Omron CX-Programmer project NewProject (CX-Programmer 9.88)

# PLC AddOn_Final_Caulking: CJ2M CPU33
I/O table (CPU CJ2M-CPU33): rack 0 slot 11 CJ2M-EIP21

## Global symbols (name address type ; comment)
W463.00 BOOL  ; PB. dispenser ON
W56.00 BOOL  ; IND. dispenser On
3205.07 BOOL  ; CR Dispenser Oil ON
AL1 H400.00 BOOL  ; AL1_EMERGENCY STOP
AL10 H400.09 BOOL  ; AL10_AIR SOURCE PS. FAULT
AL100 H406.03 BOOL  ; AL100_AS.NG PULL FAULT
AL101 H406.04 BOOL  ; AL101_NG BOX FULL
AL102 H406.05 BOOL  ; AL102_WORK FINISH FULL
AL103 H406.06 BOOL  ; AL103_SAFET DOOR IS OPEN
AL104 H406.07 BOOL  ; AL104_Positioning TImeout
AL105 H406.08 BOOL  ; AL105_
AL106 H406.09 BOOL  ; AL106_
AL107 H406.10 BOOL  ; AL107_Oil Apply UD Fault
AL108 H406.11 BOOL  ; AL108_Oil Apply AR Fault
AL109 H406.12 BOOL  ; AL109_
AL11 H400.10 BOOL  ; AL11_DUMMY DOOR OPEN
AL110 H406.13 BOOL  ; AL110_
AL111 H406.14 BOOL  ; AL111_
AL112 H406.15 BOOL  ; AL112_
AL113 H407.00 BOOL  ; AL113_
AL114 H407.01 BOOL  ; AL114_
AL115 H407.02 BOOL  ; AL115_
AL116 H407.03 BOOL  ; AL116_
AL117 H407.04 BOOL  ; AL117_
AL118 H407.05 BOOL  ; AL118_
AL119 H407.06 BOOL  ; AL119_
AL12 H400.11 BOOL  ; AL12_SHUTTER DOOR INTERRUPTED
AL120 H407.07 BOOL  ; AL120_
AL121 H407.08 BOOL  ; AL121_
AL122 H407.09 BOOL  ; AL122_
AL123 H407.10 BOOL  ; AL123_
AL124 H407.11 BOOL  ; AL124
AL125 H407.12 BOOL  ; AL125_
AL126 H407.13 BOOL  ; AL126_
AL127 H407.14 BOOL  ; AL127_
AL128 H407.15 BOOL  ; AL128:
AL129 H408.00 BOOL  ; AL129:
AL13 H400.12 BOOL  ; AL13_FNCK EMERGENCY STOP
AL130 H408.01 BOOL  ; AL130:
AL131 H408.02 BOOL  ; AL131:
AL132 H408.03 BOOL  ; AL132:
AL133 H408.04 BOOL  ; AL133:
AL134 H408.05 BOOL  ; AL134:
AL135 H408.06 BOOL  ; AL135:
AL136 H408.07 BOOL  ; AL136:
AL137 H408.08 BOOL  ; AL137:
AL138 H408.09 BOOL  ; AL138:
AL139 H408.10 BOOL  ; AL139:
AL14 H400.13 BOOL  ; AL14_FNCK FUSE ABNORMAL
AL140 H408.11 BOOL  ; AL140:
AL141 H408.12 BOOL  ; AL141:
AL142 H408.13 BOOL  ; AL142:
AL143 H408.14 BOOL  ; AL143:
AL144 H408.15 BOOL  ; AL144:
AL145 H409.00 BOOL  ; AL145:
AL146 H409.01 BOOL  ; AL146:
AL147 H409.02 BOOL  ; AL147:
AL148 H409.03 BOOL  ; AL148:
AL149 H409.04 BOOL  ; AL149:
AL15 H400.14 BOOL  ; AL15_1EC1 ABNORMAL
AL150 H409.05 BOOL  ; AL150:
AL151 H409.06 BOOL  ; AL151:
AL152 H409.07 BOOL  ; AL152:
AL153 H409.08 BOOL  ; AL153:
AL154 H409.09 BOOL  ; AL154:
AL155 H409.10 BOOL  ; AL155:
AL156 H409.11 BOOL  ; AL156:
AL157 H409.12 BOOL  ; AL157:
AL158 H409.13 BOOL  ; AL158:
AL159 H409.14 BOOL  ; AL159:
AL16 H400.15 BOOL  ; AL16_1EC2 ABNORMAL
AL160 H409.15 BOOL  ; AL160:
AL161 H410.00 BOOL  ; AL161_PRODUCTION QUANTITY WARNING
AL162 H410.01 BOOL  ; AL162_DEFECT QUANTITY WARNING
AL163 H410.02 BOOL  ; AL163_TOTAL QUANTITY WARNING
AL164 H410.03 BOOL  ; AL164_
AL165 H410.04 BOOL  ; AL165_
AL166 H410.05 BOOL  ; AL166_
AL167 H410.06 BOOL  ; AL167_
AL168 H410.07 BOOL  ; AL168_
AL169 H410.08 BOOL  ; AL169:
AL17 H401.00 BOOL  ; AL17_1EC3 ABNORMAL
AL170 H410.09 BOOL  ; AL170_WIP DISCHARGE DONE
AL171 H410.10 BOOL  ; AL171_
AL172 H410.11 BOOL  ; AL172_
AL173 H410.12 BOOL  ; AL173_
AL174 H410.13 BOOL  ; AL174_
AL175 H410.14 BOOL  ; AL175_
AL176 H410.15 BOOL  ; AL176_
AL177 H411.00 BOOL  ; AL177_
AL178 H411.01 BOOL  ; AL178_
AL179 H411.02 BOOL  ; AL179_
AL18 H401.01 BOOL  ; AL18_1EC4 ABNORMAL
AL180 H411.03 BOOL  ; AL180_
AL181 H411.04 BOOL  ; AL181_
AL182 H411.05 BOOL  ; AL182_
AL183 H411.06 BOOL  ; AL183_
AL184 H411.07 BOOL  ; AL184_
AL185 H411.08 BOOL  ; AL185_
AL186 H411.09 BOOL  ; AL186_
AL187 H411.10 BOOL  ; AL187_
AL188 H411.11 BOOL  ; AL188_
AL189 H411.12 BOOL  ; AL189_
AL19 H401.02 BOOL  ; AL19_1MTD1 ABNORMAL
AL190 H411.13 BOOL  ; AL190_
AL191 H411.14 BOOL  ; AL191_
AL192 H411.15 BOOL  ; AL192_
AL193 H412.00 BOOL  ; AL193_
AL194 H412.01 BOOL  ; AL194_
AL195 H412.02 BOOL  ; AL195_
AL196 H412.03 BOOL  ; AL196:
AL197 H412.04 BOOL  ; AL197:
AL198 H412.05 BOOL  ; AL198:
AL199 H412.06 BOOL  ; AL199:
AL2 H400.01 BOOL  ; AL2_FUSE ABNORMAL
AL20 H401.03 BOOL  ; AL20:
AL200 H412.07 BOOL  ; AL200_PLC LOW BATTERY
AL201 H412.08 BOOL  ; AL201:
AL202 H412.09 BOOL  ; AL202:
AL203 H412.10 BOOL  ; AL203:
AL204 H412.11 BOOL  ; AL204:
AL205 H412.12 BOOL  ; AL205:
AL21 H401.04 BOOL  ; AL21:
AL22 H401.05 BOOL  ; AL22:
AL23 H401.06 BOOL  ; AL23:
AL24 H401.07 BOOL  ; AL24:
AL25 H401.08 BOOL  ; AL25:
AL26 H401.09 BOOL  ; AL26:
AL27 H401.10 BOOL  ; AL27:
AL28 H401.11 BOOL  ; AL28:
AL29 H401.12 BOOL  ; AL29:
AL3 H400.02 BOOL  ; AL3_SAFETY COVER OPEN
AL30 H401.13 BOOL  ; AL30:
AL31 H401.14 BOOL  ; AL31:
AL32 H401.15 BOOL  ; AL32:
AL33 H402.00 BOOL  ; AL33_CYCLE TIME OVER
AL34 H402.01 BOOL  ; AL34_FNCK MASTER OR AUTO STOP
AL35 H402.02 BOOL  ; AL35_FNCK FAULT OCCUR
AL36 H402.03 BOOL  ; AL36_MB LOADER 1 WORK LOST
AL37 H402.04 BOOL  ; AL37_MB LOADER 2 WORK LOST
AL38 H402.05 BOOL  ; AL38_POSITIONNING UNIT WORK LOST
AL39 H402.06 BOOL  ; AL39_TRANSFER SLIDE MB LOST
AL4 H400.03 BOOL  ; AL4_AIR SOURCE LOW
AL40 H402.07 BOOL  ; AL40_DIAPHAM LOADER 1 LOST WORK
AL41 H402.08 BOOL  ; AL41_DIAPHAM LOADER 2 LOST WORK
AL42 H402.09 BOOL  ; AL42_DIAPHAM LOADER 3 LOST WORK
AL43 H402.10 BOOL  ; AL43_DIAPHAM VACCUM STATION WORK LOST
AL44 H402.11 BOOL  ; AL44_DIAPHAM BUFFER STATION WORK LOST
AL45 H402.12 BOOL  ; AL45_DIAPHAM FEED IN STATION ABNORMAL
AL46 H402.13 BOOL  ; AL46_TRANFER SLIDE DIAPHAM LOST
AL47 H402.14 BOOL  ; AL47_ROTARY GRIPPER 1 LOST WORK
AL48 H402.15 BOOL  ; AL48_ROTARY GRIPPER 2 LOST WORK
AL49 H403.00 BOOL  ; AL49_WORK DISCHARGE UNIT WORK LOST
AL5 H400.04 BOOL  ; AL5_DEVICE-NET FAULT
AL50 H403.01 BOOL  ; AL50:Work Floating
AL51 H403.02 BOOL  ; AL51:
AL52 H403.03 BOOL  ; AL52:
AL53 H403.04 BOOL  ; AL53:
AL54 H403.05 BOOL  ; AL54:
AL55 H403.06 BOOL  ; AL55:
AL56 H403.07 BOOL  ; AL56:
AL57 H403.08 BOOL  ; AL57:
AL58 H403.09 BOOL  ; AL58:
AL59 H403.10 BOOL  ; AL59:
AL6 H400.05 BOOL  ; AL6_PLC ABNORMAL
AL60 H403.11 BOOL  ; AL60:
AL61 H403.12 BOOL  ; AL61:
AL62 H403.13 BOOL  ; AL62:
AL63 H403.14 BOOL  ; AL63:
AL64 H403.15 BOOL  ; AL64:
AL65 H404.00 BOOL  ; AL65_PRODUCTION QUANTITY UP
AL66 H404.01 BOOL  ; AL66_DEFECT QUANTITY UP
AL67 H404.02 BOOL  ; AL67_TOTAL QUANTITY UP
AL68 H404.03 BOOL  ; AL68_
AL69 H404.04 BOOL  ; AL69_
AL7 H400.06 BOOL
AL70 H404.05 BOOL  ; AL70_
AL71 H404.06 BOOL  ; AL71_
AL72 H404.07 BOOL  ; AL72_
AL73 H404.08 BOOL
AL74 H404.09 BOOL
AL75 H404.10 BOOL
AL76 H404.11 BOOL
AL77 H404.12 BOOL
AL78 H404.13 BOOL
AL79 H404.14 BOOL
AL8 H400.07 BOOL
AL80 H404.15 BOOL
AL81 H405.00 BOOL  ; AL81_AS.SHUTTER 1 FAULT
AL82 H405.01 BOOL  ; AL82_AS.SHUTTER 2 FAULT
AL83 H405.02 BOOL  ; AL83_AS.DIAPH GRIPPER UNIT FAULT
AL84 H405.03 BOOL  ; AL84_AS.DIAPH GRIPPER 1 FAULT
AL85 H405.04 BOOL  ; AL85_AS.DIAPH GRIPPER 2 FAULT
AL86 H405.05 BOOL  ; AL86_AS.DIAPH GRIPPER 3 FAULT
AL87 H405.06 BOOL  ; AL87_AS.DIAPH GRIPPER FLIP FAULT
AL88 H405.07 BOOL  ; AL88_AS.ROTARY GRIPPER 1 FAULT
AL89 H405.08 BOOL  ; AL89_AS.ROTARY GRIPPER 2 FAULT
AL9 H400.08 BOOL
AL90 H405.09 BOOL  ; AL90_AS.ROTARY GRIPPER UNIT 1 FAULT
AL91 H405.10 BOOL  ; AL91_AS.ROTARY GRIPPER UNIT 2 FAULT
AL92 H405.11 BOOL  ; AL92_AS.MB LOAD IN FAULT
AL93 H405.12 BOOL  ; AL93_AS.MB LOAD OUT FAULT
AL94 H405.13 BOOL  ; AL94_AS.MB LOAD OUT UNIT FAULT
AL95 H405.14 BOOL  ; AL95_AS.MB SLIDE UNIT FAULT
AL96 H405.15 BOOL  ; AL96_AS.MB POSITION PIN UNIT FAULT
AL97 H406.00 BOOL  ; AL97_AS.WORK TRANSFER UNIT FAULT
AL98 H406.01 BOOL  ; AL98_AS.FINISH TRAY FAULT
AL99 H406.02 BOOL  ; AL99_AS.OK PUSH FAULT
ALMF001 W501.00 BOOL  ; ALMF001_SHUTTER 1 OPERATION FAULT
ALMF002 W501.01 BOOL  ; ALMF002_SHUTTER 2 OPERATION FAULT
ALMF003 W501.02 BOOL  ; ALMF003_DIAPH GRIPPER UNIT OPERATION FAULT
ALMF004 W501.03 BOOL  ; ALMF004_DIAPH GRIPPER 1 OPERATION FAULT
ALMF005 W501.04 BOOL  ; ALMF005_DIAPH GRIPPER 2 OPERATION FAULT
ALMF006 W501.05 BOOL  ; ALMF006_DIAPH GRIPPER 3 OPERATION FAULT
ALMF007 W501.06 BOOL  ; ALMF007_DIAPH GRIPPER FLIP OPERATION FAULT
ALMF008 W501.07 BOOL  ; ALMF008_ROTARY GRIPPER 1 OPERATION FAULT
ALMF009 W501.08 BOOL  ; ALMF009_ROTARY GRIPPER 2 OPERATION FAULT
ALMF010 W501.09 BOOL  ; ALMF010_ROTARY GRIPPER UNIT 1 OPERATION FAULT
ALMF011 W501.10 BOOL  ; ALMF011_ROTARY GRIPPER UNIT 2 OPERATION FAULT
ALMF012 W501.11 BOOL  ; ALMF012_MB LOAD IN OPERATION FAULT
ALMF013 W501.12 BOOL  ; ALMF013_MB LOAD OUT OPERATION FAULT
ALMF014 W501.13 BOOL  ; ALMF014_MB LOAD OUT UNIT OPERATION FAULT
ALMF015 W501.14 BOOL  ; ALMF015_MB SLIDE UNIT OPERATION FAULT
ALMF016 W501.15 BOOL  ; ALMF016_MB POSITION PIN UNIT OPERATION FAULT
ALMF017 W502.00 BOOL  ; ALMF017_WORK TRANSFER UNIT OPERATION FAULT
ALMF018 W502.01 BOOL  ; ALMF018_FINISH TRAY OPERATION FAULT
ALMF019 W502.02 BOOL  ; ALMF019_OK PUSH OPERATION FAULT
ALMF020 W502.03 BOOL  ; ALMF020_NG PULL OPERATION FAULT
0.00 BOOL  ; PB.EMG STOP
0.01 BOOL  ; AIR SOURCE CONF.
0.02 BOOL  ; SS.AUTO-IND.(AUTO=ON)
0.03 BOOL  ; PB.MASTER ON
0.04 BOOL  ; PB.AUTO RUN
0.05 BOOL  ; PB.CYCLE STOP
0.06 BOOL  ; PB.DUMMY DOOR OPEN REQUEST
0.07 BOOL  ; CR.TEACHING ON
0.08 BOOL  ; CR.MACHINR DOOR CONFIRM
0.09 BOOL  ; CR.DUMMY DOOR CONFIRM
0.10 BOOL  ; CR.SHUTTER DOOR OUT CONFIRM
0.11 BOOL  ; CR.SHUTTER DOOR IN CONFIRM
0.12 BOOL  ; CR.MASTER ON CONFIRM
0.13 BOOL  ; CR.FUSE NORMAL CONFIRM
0.14 BOOL  ; CR.DIAPHAM DOOR ENABLE CONF
0.15 BOOL  ; .
1516 CHANNEL  ; SLAVE STATUS 1
1517 CHANNEL  ; SLAVE STATUS 2
1518 CHANNEL  ; SLAVE STATUS 3
1519 CHANNEL  ; SLAVE STATUS 4
1520 CHANNEL  ; NORMAL SLAVE1
1522 CHANNEL  ; NORMAL SLAVE3
1541 CHANNEL  ; SLAVE STATUS 1
1542 CHANNEL  ; SLAVE STATUS 2
1543 CHANNEL  ; SLAVE STATUS 3
1544 CHANNEL  ; SLAVE STATUS 4
1545 CHANNEL  ; NORMAL SLAVE STATUS 1
1547 CHANNEL  ; NORMAL SLAVE STATUS 3
1.00 BOOL  ; CR.EMERGENCY STOP INTERLOCK
1.01 BOOL  ; PL.AUTO RUNNING
1.02 BOOL  ; PL.MASTER ON
1.03 BOOL  ; PL.OK TO FEED DIAPHAM
1.04 BOOL  ; PL.DUMMY DOOR ENABLE CONFIRM
1.05 BOOL  ; PL.DUMMY PROCESS
1.06 BOOL  ; BZ.BUZZER
1.07 BOOL  ; CR.ADD-ON ABNORMAL INTERLOCK
1.08 BOOL  ; CR.ADD-ON AUTO RUN INTERLOCK
1.09 BOOL  ; CR.DUMMY DOOR ENABLE TO OPEN
1.10 BOOL  ; CR Interupt Safety area
1.11 BOOL  ; CR.TEACHING ENABLE
1.12 BOOL  ; CR.ADD-ON AUTO START
1.13 BOOL  ; PL.SIGNAL TOWER R
1.14 BOOL  ; PL.SIGNAL TOWER Y
1.15 BOOL  ; PL.SIGNAL TOWER G
2.00 BOOL  ; ITLK.PB FINAL EMERGENCY NOT
2.01 BOOL  ; ITLK.FINAL CAULKING FUSE CONFIRM
2.02 BOOL  ; ITLK.FINAL CAULKING-MASTER ON,AUTO RUNNING
2.03 BOOL  ; ITLK.FINAL CAULKING-ALL HOME
2.04 BOOL  ; ITLK.FINAL CAULKING DIAPH BLOW OK
2.05 BOOL  ; ITLK.FINAL CAULKING ABNORMAL DETECTION
2.06 BOOL  ; .
2.07 BOOL  ; ITLK.FINAL CAULKING-AUTO M&B VACCUM OK
2.08 BOOL  ; ITLK.FINAL CAULKING-AUTO DIAPH VACCUM OK
2.09 BOOL  ; ITLK.FINAL CAULKING WORK OK
2.10 BOOL  ; ITLK.FINAL CAULKING WORK NG
2.11 BOOL  ; ITLK.FINAL CAULKING WORK OPERATE
2.12 BOOL  ; ITLK.PH FINAL CAULKING ST1 DETECT
2.13 BOOL  ; ITLK.PH FINAL CAULKING ST2 DETECT
2.14 BOOL  ; .
2.15 BOOL  ; .
3205.00 BOOL  ; 1MTD1.FWD
3205.01 BOOL  ; 1MTD1.REV
3205.02 BOOL  ; 1MTD1.MO
3205.03 BOOL  ; 1MGH1 START
3205.04 BOOL  ; 1MGH1 STOP
3205.05 BOOL  ; 1MGH2 START
3205.06 BOOL  ; 1MGH2 STOP
3205.08 BOOL  ; SOL. SHUTTER DOOR 1 DOWN
3205.09 BOOL  ; SOL. SHUTTER DOOR 2 UP
3205.10 BOOL  ; SOL. SHUTTER DOOR 2 DOWN
3205.15 BOOL  ; PL.LOAD WORK ENABLE
3207.00 BOOL  ; SOL_Oil Apply Ret
3207.01 BOOL  ; SOL_Oil Apply Adv
3207.02 BOOL  ; SOL_Oil Apply Down
3207.03 BOOL  ; SOL_Oil Apply Up
3211.00 BOOL  ; M&B LOAD UNIT SLIDE ADV
3211.01 BOOL  ; M&B LOAD UNIT SLIDE RET
3211.02 BOOL  ; M&B LOAD IN DOWN
3211.03 BOOL  ; M&B LOAD IN UP
3211.04 BOOL  ; M&B LOAD OUT UNIT DOWN
3211.05 BOOL  ; M&B LOAD OUT UNIT UP
3211.06 BOOL  ; M&B LOAD OUT DOWN
3211.07 BOOL  ; M&B LOAD OUT UP
3211.08 BOOL  ; PIN POSIRIONNING UP
3211.09 BOOL  ; PIN POSIRIONNING DOWN
3211.10 BOOL  ; NG PUSH DOWN
3211.11 BOOL  ; NG PUSH UP
3211.12 BOOL  ; OK PUSH UP
3211.13 BOOL  ; OK PUSH DOWN
3211.14 BOOL  ; LOAD BWD
3211.15 BOOL  ; LOAD FWD
3213.00 BOOL  ; WORK FINISH TRAY DOWN CONFIRM
3213.01 BOOL  ; WORK FINISH TRAY UP CONFIrM
3213.02 BOOL  ; TRANSFER SLIDE UNIT ADV
3213.03 BOOL  ; TRANSFER SLIDE UNIT RET
3213.04 BOOL  ; GIPPER TRANSFER UNIT 1 UNIT ADV
3213.05 BOOL  ; GIPPER TRANSFER UNIT 1 UNIT RET
3213.06 BOOL  ; GIPPER TRANSFER UNIT 2 UNIT ADV
3213.07 BOOL  ; GIPPER TRANSFER UNIT 2 UNIT RET
3213.08 BOOL  ; GIPPER TRANSFER 1 UNIT CHUCK
3213.09 BOOL  ; GIPPER TRANSFER 1 UNIT UNCHUCK
3213.10 BOOL  ; GIPPER TRANSFER 2 UNIT CHUCK
3213.11 BOOL  ; GIPPER TRANSFER 2 UNIT UNCHUCK
3213.12 BOOL  ; .
3213.13 BOOL  ; .
3213.14 BOOL  ; .
3213.15 BOOL  ; .
3215.00 BOOL  ; GRIPPER UNIT DOWN
3215.01 BOOL  ; GRIPPER UNIT UP
3215.02 BOOL  ; GRIPPER 1 DIAPH CHUCK
3215.03 BOOL  ; GRIPPER 1 DIAPH UNCHUCK
3215.04 BOOL  ; GRIPPER 2 DIAPH CHUCK
3215.05 BOOL  ; GRIPPER 2 DIAPH UNCHUCK
3215.06 BOOL  ; FLIP DIAPH 180
3215.07 BOOL  ; FLIP DIAPH 0
3215.08 BOOL  ; GRIPPER 3 DIAPH CHUCK
3215.09 BOOL  ; GRIPPER 3 DIAPH UNCHUCK
3215.10 BOOL  ; .
3215.11 BOOL  ; .
3215.12 BOOL  ; .
3215.13 BOOL  ; .
3215.14 BOOL  ; .
3215.15 BOOL  ; .
3301.00 BOOL  ; AS.SHUTTER 1 DOOR UP CONFIRM
3301.01 BOOL  ; AS.SHUTTER 1 DOOR DOWN CONFIRM
3301.02 BOOL  ; AS.SHUTTER 2 DOOR UP CONFIRM
3301.03 BOOL  ; AS.SHUTTER 2 DOOR DOWN CONFIRM
3301.04 BOOL  ; AS.GRIPPER UNIT DOWN CONFIRM
3301.05 BOOL  ; AS.GRIPPER UNIT UP CONFIRM
3301.06 BOOL  ; AS.GRIPPER 1 DIAPH CHUCK. CONFIRM
3301.07 BOOL  ; AS.GRIPPER 1 DIAPH UNCHUCK. CONFIRM
3301.08 BOOL  ; AS.GRIPPER 2 DIAPH CHUCK. CONFIRM
3301.09 BOOL  ; AS.GRIPPER 2 DIAPH UNCHUCK. CONFIRM
3301.10 BOOL  ; AS.GRIPPER 3 DIAPH CHUCK. CONFIRM
3301.11 BOOL  ; AS.GRIPPER 3 DIAPH UNCHUCK. CONFIRM
3301.12 BOOL  ; AS.FLIP DIAPH 180. CONFIRM
3301.13 BOOL  ; AS.FLIP DIAPH 0. CONFIRM
3301.14 BOOL  ; 1MTD1.ALARM
3301.15 BOOL  ; AUTO START(NAGARA)
3302.00 BOOL  ; AS.GIPPER TRANSFER 1 UNIT CHUCK CONFIRM
3302.01 BOOL  ; AS.GIPPER TRANSFER 1 UNIT  UNCHUCK CONFIRM
3302.02 BOOL  ; AS.GIPPER TRANSFER 2 UNIT CHUCK CONFIRM
3302.03 BOOL  ; AS.GIPPER TRANSFER 2 UNIT  UNCHUCK CONFIRM
3302.04 BOOL  ; AS.GIPPER TRANSFER UNIT 1 UNIT ADV. CONFIRM
3302.05 BOOL  ; AS.GIPPER TRANSFER UNIT 1 UNIT RET. CONFIRM
3302.06 BOOL  ; AS.GIPPER TRANSFER UNIT 2 UNIT ADV. CONFIRM
3302.07 BOOL  ; AS.GIPPER TRANSFER UNIT 2 UNIT RET. CONFIRM
3302.08 BOOL  ; PH MB VAcuum
3302.09 BOOL  ; PH. WORK FULL
3302.10 BOOL  ; PH.TRANSFER STATION DIAPH SIDE CONFIRM
3302.11 BOOL  ; PH.TRANSFER STATION DIAPH WORK CONFIRM
3302.12 BOOL  ; PH.TRANSFER STATION M&B WORK CONFIRM
3302.13 BOOL  ; PH. M&B LOADER WORK CONF 1
3302.14 BOOL  ; PH. M&B LOADER WORK CONF 2
3302.15 BOOL  ; PH. WORK IN ROTATE UNIT CONFIRM
3303.00 BOOL  ; AS.M&B LOAD IN DOWN.CONFIRM
3303.01 BOOL  ; AS.M&B LOAD IN UP.CONFIRM
3303.02 BOOL  ; AS.M&B LOAD OUT DOWN.CONFIRM
3303.03 BOOL  ; AS.M&B LOAD OUT UP.CONFIRM
3303.04 BOOL  ; AS.M&B LOAD OUT UNIT DOWN.CONFIRM
3303.05 BOOL  ; AS.M&B LOAD OUT UNIT UP.CONFIRM
3303.06 BOOL  ; AS.M&B LOAD UNIT SLIDE ADV.CONFIRM
3303.07 BOOL  ; AS.M&B LOAD UNIT SLIDE RET.CONFIRM
3303.08 BOOL  ; AS.PIN POSIRIONNING UP CONFIRM
3303.09 BOOL  ; AS.PIN POSIRIONNING DOWN CONFIRM
3303.10 BOOL  ; AS.TRANSFER SLIDE UNIT ADV. CONFIRM
3303.11 BOOL  ; AS.TRANSFER SLIDE UNIT RET. CONFIRM
3303.12 BOOL  ; PH work infinish tray
3303.13 BOOL  ; .
3303.14 BOOL  ; AS LOAD BWD
3303.15 BOOL  ; AS LOAD FWD
3304.00 BOOL  ; AS.WORK FINISH TRAY DOWN CONFIRM
3304.01 BOOL  ; AS.WORK FINISH TRAY UP CONFIRM
3304.02 BOOL  ; AS.OK PUSH UP. CONFIRM
3304.03 BOOL  ; AS.OK PUSH DOWN. CONFIRM
3304.04 BOOL  ; AS.NG PUSH DOWN. CONFIRM
3304.05 BOOL  ; AS.NG PUSH UP. CONFIRM
3304.06 BOOL  ; .
3304.07 BOOL  ; temporary nagara
3304.08 BOOL  ; PH. WORK ROTATE PRE-END CONFIRM
3304.09 BOOL  ; PH. TEMINAL IN POSITION CONFIRM
3304.10 BOOL  ; PH. WORK DIAPH LOAD IN CONFIRM
3304.11 BOOL  ; PH.STATION DIAPH VACCUM CONFIRM
3304.12 BOOL  ; PH.STATION BUFFER DIAPH CONFIRM
3304.13 BOOL  ; PH. WORK NG CONFIRM
3304.14 BOOL  ; PH. WORK OK CONFIRM
3304.15 BOOL  ; Safety AREA
3307.00 BOOL  ; RS_Oil Apply DOWN
3307.01 BOOL  ; RS_Oil Apply UP
3307.02 BOOL  ; RS_Oil Apply ADV
3307.03 BOOL  ; RS_Oil Apply RET
3334.01 BOOL  ; AS.WORK FINISH TRAY UP CONFIRM
3356.01 BOOL  ; diap auto
370.10 BOOL  ; PL HMI CAULKING ST1
370.11 BOOL  ; PL Rotary Gipper 2
370.12 BOOL  ; PL rotary gripper 1
370.13 BOOL  ; PL OKNG disch
3.00 BOOL  ; 1EC1.FORWARD START (DOWN)
3.01 BOOL  ; 1EC1.BACKWARD START (UP)
3.02 BOOL  ; 1EC1.ALARM RESET
3.03 BOOL  ; 1EC1.BREAK RELEASE (MTN)
3.04 BOOL  ; 1EC2.FWD START
3.05 BOOL  ; 1EC2.BWD START
3.06 BOOL  ; 1EC2.ALARM RESET
3.07 BOOL  ; 1EC2.BREAK RELEASE (MTN)
3.08 BOOL  ; 1EC3.FORWARD START
3.09 BOOL  ; 1EC3.BACKWARD START
3.10 BOOL  ; 1EC3.ALARM RESET
3.11 BOOL  ; 1EC3.BREAK RELEASE (MTN)
3.12 BOOL  ; 1EC4.FORWARD START
3.13 BOOL  ; 1EC4.BACKWARD START
3.14 BOOL  ; 1EC4.ALARM RESET
3.15 BOOL  ; 1EC4.BREAK RELEASE (MTN)
4450.00 BOOL  ; PB triall mode
4460.00 BOOL  ; PL trial mode
4.00 BOOL  ; 1EC1.FORWARD COMPLETE
4.01 BOOL  ; 1EC1.BACKWARD COMPLETE
4.02 BOOL  ; 1EC1.ALARM
4.03 BOOL  ; 1EC2.FORWARD COMPLETE
4.04 BOOL  ; 1EC2.BACKWARD COMPLETE
4.05 BOOL  ; 1EC2.ALARM
4.06 BOOL  ; 1EC3.FORWARD COMPLETE
4.07 BOOL  ; 1EC3.BACKWARD COMPLETE
4.08 BOOL  ; 1EC3.MIDDLE COMPLETE
4.09 BOOL  ; .
4.10 BOOL  ; .
4.11 BOOL  ; 1EC4.BACKWARD COMPLETE
4.12 BOOL  ; 1EC4.ALARM
4.15 BOOL  ; Safety area
56.06 BOOL  ; TIMER
5.00 BOOL  ; DIAPHAM DOOR ENABLE
5.01 BOOL  ; IAI EC POWER
5.05 BOOL  ; MG1 ON
5.06 BOOL  ; mg 1 off
5.07 BOOL  ; mg 2 on
5.08 BOOL  ; mg2 off
999.00 BOOL  ; ASAKE MODIFY (Oil Apply)
A202.00 BOOL  ; Communications Port Enabled Flag, Port No. 0
A202.01 BOOL  ; Communications Port Enabled Flag, Port No. 1
A202.02 BOOL  ; Communications Port Enabled Flag, Port No. 2
A202.03 BOOL  ; Communications Port Enabled Flag, Port No. 3
A202.04 BOOL  ; Communications Port Enabled Flag, Port No. 4
A202.05 BOOL  ; Communications Port Enabled Flag, Port No. 5
A202.06 BOOL  ; Communications Port Enabled Flag, Port No. 6
A202.07 BOOL  ; Communications Port Enabled Flag, Port No. 7
A401.10 BOOL  ; I/O_SETTING FAULT FLAG
A401.11 BOOL  ; I/O_MARK OVER FLAG
A401.13 BOOL  ; No.DOBLE USE FAULT FLAG
A401.14 BOOL  ; I/O BUS FAULT FLAG
A401.15 BOOL  ; MEMORY FAULT FLAG
A402.02 BOOL  ; High performance I/O unit setting and abnormality flags
A402.03 BOOL  ; CPU high performance unit setting and abnormality flags
A402.07 BOOL  ; High performance I unit of CPU abnormal flag
C0401 BOOL  ; CT01_LOW_UP
C0402 BOOL  ; CT01_HI_UP
C0403 BOOL  ; CT02_LOW_UP
C0404 BOOL  ; CT02_HI_UP
C0405 BOOL  ; CT03_LOW_UP
C0406 BOOL  ; CT03_HI_UP
C0407 BOOL  ; CT04_LOW_UP
C0408 BOOL  ; CT04_HI_UP
C0409 BOOL  ; CT05_LOW_UP
C0410 BOOL  ; CT05_HI_UP
C0411 BOOL  ; CT06_LOW_UP
C0412 BOOL  ; CT06_HI_UP
C0413 BOOL  ; CT07_LOW_UP
C0414 BOOL  ; CT07_HI_UP
C0415 BOOL  ; CT08_LOW_UP
C0416 BOOL  ; CT08_HI_UP
C0417 BOOL  ; CT09_LOW_UP
C0418 BOOL  ; CT09_HI_UP
C0419 BOOL  ; CT10_LOW_UP
C0420 BOOL  ; CT10_HI_UP
C0421 BOOL  ; CT11_LOW_UP
C0422 BOOL  ; CT11_HI_UP
C0423 BOOL  ; CT12_LOW_UP
C0424 BOOL  ; CT12_HI_UP
C0425 BOOL  ; CT13_LOW_UP
C0426 BOOL  ; CT13_HI_UP
C0427 BOOL  ; CT14_LOW_UP
C0428 BOOL  ; CT14_HI_UP
C0429 BOOL  ; CT15_LOW_UP
C0430 BOOL  ; CT15_HI_UP
C0451 BOOL  ; T1_LOW_UP
C0453 BOOL  ; T2_LOW_UP
C0455 BOOL  ; T3_LOW_UP
C0457 BOOL  ; T4_LOW_UP
C0459 BOOL  ; T5_LOW_UP
C0461 BOOL  ; T6_LOW_UP
C0468 BOOL  ; MONITORING CT_LOW
C0472 BOOL  ; AUTOMATIC TIME S
C0473 BOOL  ; AUTOMATIC TIME M
C0474 BOOL  ; AUTOMATIC TIME H
C0475 BOOL  ; WAITING-TIME S
C0476 BOOL  ; WAITING-TIME M
C0478 BOOL  ; STOP TIME S
C0479 BOOL  ; STOP TIME M
C0501 BOOL  ; OUTPUT 1 CUMULATE TIME m
C0502 BOOL  ; OUTPUT 2 CUMULATE TIME m
C0503 BOOL  ; OUTPUT 3 CUMULATE TIME m
C0504 BOOL  ; OUTPUT 4 CUMULATE TIME m
C0505 BOOL  ; OUTPUT 5 CUMULATE TIME m
C401 CHANNEL  ; CT01_LOW
C402 CHANNEL  ; CT01_HI
C403 CHANNEL  ; CT02_LOW
C404 CHANNEL  ; CT02_HI
C405 CHANNEL  ; CT03_LOW
C406 CHANNEL  ; CT03_HI
C407 CHANNEL  ; CT04_LOW
C408 CHANNEL  ; CT04_HI
C409 CHANNEL  ; CT05_LOW
C410 CHANNEL  ; CT05_HI
C411 CHANNEL  ; CT06_LOW
C412 CHANNEL  ; CT06_HI
C413 CHANNEL  ; CT07_LOW
C414 CHANNEL  ; CT07_HI
C415 CHANNEL  ; CT08_LOW
C416 CHANNEL  ; CT08_HI
C417 CHANNEL  ; CT09_LOW
C418 CHANNEL  ; CT09_HI
C419 CHANNEL  ; CT10_LOW
C420 CHANNEL  ; CT10_HI
C421 CHANNEL  ; CT11_LOW
C422 CHANNEL  ; CT11_HI
C423 CHANNEL  ; CT12_LOW
C424 CHANNEL  ; CT12_HI
C425 CHANNEL  ; CT13_LOW
C426 CHANNEL  ; CT13_HI
C427 CHANNEL  ; CT14_LOW
C428 CHANNEL  ; CT14_HI
C429 CHANNEL  ; CT15_LOW
C430 CHANNEL  ; CT15_HI
C451 CHANNEL  ; T1_LOW
C452 CHANNEL  ; T1_HI
C453 CHANNEL  ; T2_LOW
C454 CHANNEL  ; T2_HI
C455 CHANNEL  ; T3_LOW
C456 CHANNEL  ; T3_HI
C457 CHANNEL  ; T4_LOW
C458 CHANNEL  ; T4_HI
C459 CHANNEL  ; T5_LOW
C460 CHANNEL  ; T5_HI
C461 CHANNEL  ; T6_LOW
C462 CHANNEL  ; T6_HI
C501 CHANNEL  ; OUTPUT 1 CUMULATE TIME m
C502 CHANNEL  ; OUTPUT 2 CUMULATE TIME m
C503 CHANNEL  ; OUTPUT 3 CUMULATE TIME m
C504 CHANNEL  ; OUTPUT 4 CUMULATE TIME m
C505 CHANNEL  ; OUTPUT 5 CUMULATE TIME m
D1 CHANNEL  ; MB Loader Work Grip
D100 CHANNEL  ; SUM MB AUX1
D101 CHANNEL  ; SUM ALL MB
D110 CHANNEL  ; AUX1
D111 CHANNEL  ; AUX2
D112 CHANNEL  ; AUX3
D113 CHANNEL  ; WORK DIAPHAM +1
D114 CHANNEL  ; DIAPH SUMMARY
D12 CHANNEL  ; MB Rotate Work
D200 CHANNEL  ; WORK LAST ORER
D2000 CHANNEL  ; MB LOAD IN TIMER
D201 CHANNEL  ; WORK FEED OUT
D202 CHANNEL  ; LAST ORDER COUNT FOR P16
D22 CHANNEL  ; TRANSFER WORK
D23 CHANNEL  ; TRANSFER WORK
D3000 CHANNEL  ; DATA PASSWORD FROM SREEN
D3004 CHANNEL  ; DATA PASS WORD CHECK USE
D3020 CHANNEL  ; OFFSET ANGLE HMI
D3024 CHANNEL  ; OFFSET ANGLE USE
D3030 CHANNEL  ; DATA ANGLE NEW OFFSET
D32 CHANNEL  ; WORK FEED IN
D3500 CHANNEL  ; DATA MM/DD (HEX)
D3502 CHANNEL  ; DATA YYYY (HEX)
D3504 CHANNEL  ; DATA MM/DD (ASC)
D3512 CHANNEL  ; DATA YYYY ASCII
D3520 CHANNEL  ; DATA YYYY(ASCII)
D4000 CHANNEL  ; No.WORD SUM CHECK
D4001 CHANNEL  ; CONTROL DATA 2
D41 CHANNEL  ; DPH Loader GRIP
D4100 CHANNEL  ; TOURQE CHECK +NG
D4102 CHANNEL  ; TOURQE CHECK -NG
D4104 CHANNEL  ; ANGLE CHECK +NG
D4106 CHANNEL  ; ANGLE CHECK -NG
D42 CHANNEL  ; DPH Loader BUFF
D5000 CHANNEL  ; VT PAGE MONITOR
D5002 CHANNEL  ; VT PAGE CONTROL
D5003 CHANNEL  ; VT SCREEN ON-OFF
D5006 CHANNEL  ; OPERATION MONITORING OUTPUT
D5011 CHANNEL  ; OPERATION MONITORING TRANSMISSION
D5013 CHANNEL  ; OPERATION MONITORING TRANSMISSION
D5047 CHANNEL  ; COMPLETED CHECK
D5049 CHANNEL  ; WATCH_DOG_HEXFF
D5066 CHANNEL  ; CYCLE TIME
D5100 CHANNEL  ; CYCLE TIME SETTING (LOW RANK)
D5101 CHANNEL  ; ACTIVE-TIME H SETTING (LOW RANK)
D5102 CHANNEL  ; ACTIVE-TIME M SETTING (LOW RANK)
D5103 CHANNEL  ; PLAN TIME H SETTING (LOW RANK)
D5104 CHANNEL  ; PLAN TIME M SETTING (LOW RANK)
D5105 CHANNEL  ; QUANTITY (LOW RANK)
D5106 CHANNEL  ; QUANTITY (HIGHER RANK)
D5108 CHANNEL  ; AUTOMATIC TIME M
D5109 CHANNEL  ; AUTOMATIC TIME H
D5111 CHANNEL  ; WAITING-TIME M
D5113 CHANNEL  ; STOP TIME M
D5120 CHANNEL  ; FAULT CHECK
D5121 CHANNEL  ; MOTION FAULT CHECK
D5131 CHANNEL  ; CT01 COUNTER
D5133 CHANNEL  ; CT02 COUNTER
D5135 CHANNEL  ; CT03 COUNTER
D5137 CHANNEL  ; CT04 COUNTER
D5139 CHANNEL  ; CT05 COUNTER
D5141 CHANNEL  ; CT06 COUNTER
D5143 CHANNEL  ; CT07 COUNTER
D5145 CHANNEL  ; CT08 COUNTER
D5147 CHANNEL  ; CT09 COUNTER
D5149 CHANNEL  ; CT10 COUNTER
D5151 CHANNEL  ; CT11 COUNTER
D5153 CHANNEL  ; CT12 COUNTER
D5155 CHANNEL  ; CT13 COUNTER
D5157 CHANNEL  ; CT14 COUNTER
D5159 CHANNEL  ; CT15 COUNTER
D5231 CHANNEL  ; CT01 COUNTER
D5341 CHANNEL  ; OUTPUT 1 START DELAY TIME
D5342 CHANNEL  ; OUTPUT 2 START DELAY TIME
D5343 CHANNEL  ; OUTPUT 3 START DELAY TIME
D5344 CHANNEL  ; OUTPUT 4 START DELAY TIME
D5345 CHANNEL  ; OUTPUT 5 START DELAY TIME
D5351 CHANNEL  ; OUTPUT 1 BREAK DELAY TIME
D5352 CHANNEL  ; OUTPUT 2 BREAK DELAY TIME
D5353 CHANNEL  ; OUTPUT 3 BREAK DELAY TIME
D5354 CHANNEL  ; OUTPUT 4 BREAK DELAY TIME
D5355 CHANNEL  ; OUTPUT 5 BREAK DELAY TIME
D5461 CHANNEL  ; OUTPUT 1 STOP SELECTION
D5462 CHANNEL  ; OUTPUT 2 STOP SELECTION
D5463 CHANNEL  ; OUTPUT 3 STOP SELECTION
D5464 CHANNEL  ; OUTPUT 4 STOP SELECTION
D5465 CHANNEL  ; OUTPUT 5 STOP SELECTION
D5471 CHANNEL  ; OUTPUT 1 EXTERNAL PRESENCE SEL.
D5472 CHANNEL  ; OUTPUT 2 EXTERNAL PRESENCE SEL.
D5473 CHANNEL  ; OUTPUT 3 EXTERNAL PRESENCE SEL.
D5474 CHANNEL  ; OUTPUT 4 EXTERNAL PRESENCE SEL.
D5475 CHANNEL  ; OUTPUT 5 EXTERNAL PRESENCE SEL.
D5481 CHANNEL  ; OUTPUT 1 LOW ENERGY TIME
D5482 CHANNEL  ; OUTPUT 2 LOW ENERGY TIME
D5483 CHANNEL  ; OUTPUT 3 LOW ENERGY TIME
D5484 CHANNEL  ; OUTPUT 4 LOW ENERGY TIME
D5485 CHANNEL  ; OUTPUT 5 LOW ENERGY TIME
D5486 CHANNEL  ; OUTPUT 1 START DELAY TIME(BIN)
D5487 CHANNEL  ; OUTPUT 2 START DELAY TIME(BIN)
D5488 CHANNEL  ; OUTPUT 3 START DELAY TIME(BIN)
D5489 CHANNEL  ; OUTPUT 4 START DELAY TIME(BIN)
D5490 CHANNEL  ; OUTPUT 5 START DELAY TIME(BIN)
D5491 CHANNEL  ; OUTPUT 1 LOW ENERGY TIME(BIN)
D5492 CHANNEL  ; OUTPUT 2 LOW ENERGY TIME(BIN)
D5493 CHANNEL  ; OUTPUT 3 LOW ENERGY TIME(BIN)
D5494 CHANNEL  ; OUTPUT 4 LOW ENERGY TIME(BIN)
D5495 CHANNEL  ; OUTPUT 5 LOW ENERGY TIME(BIN)
D5496 CHANNEL  ; OUTPUT 1 BREAK DELAY TIME(BIN)
D5497 CHANNEL  ; OUTPUT 2 BREAK DELAY TIME(BIN)
D5498 CHANNEL  ; OUTPUT 3 BREAK DELAY TIME(BIN)
D5499 CHANNEL  ; OUTPUT 4 BREAK DELAY TIME(BIN)
D5500 CHANNEL  ; OUTPUT 5 BREAK DELAY TIME(BIN)
D5600 CHANNEL  ; WORK INFO
D6000 CHANNEL  ; FIRST ID DATA READ
D6003 CHANNEL  ; SUM CHECK
D6004 CHANNEL  ; SOURCE FIRST DATA
D6006 CHANNEL  ; SERAIL No. FROM ID
D6008 CHANNEL  ; PART No. FROM ID
D6009 CHANNEL  ; PROCESS COMPLETE 1 READ FORM ID
D6010 CHANNEL  ; PROCESS COMPLETE MC.No.2 READ FORM ID
D6011 CHANNEL  ; PROCESS OK 1 FROM ID
D6013 CHANNEL  ; WORK INFO
D6031 CHANNEL  ; FINAL ID DATA READ
D6205 CHANNEL  ; TORQUE DATA 1st STAGE (ARRANGED)
D6206 CHANNEL  ; ANGLE DATA 1st STAGE (ARRANGED)
D6207 CHANNEL  ; SNUG TORQUE 1st STAGE (ARRANGED)
D6208 CHANNEL  ; TORQUE DATA 2nd STAGE (ARRANGED)
D6209 CHANNEL  ; ANGLE DATA 2nd STAGE (ARRANGED)
D6210 CHANNEL  ; SNUG TORQUE 2nd STAGE (ARRANGED)
D6211 CHANNEL  ; T/R1 2nd STAGE (ARRANGED)
D6212 CHANNEL  ; T/R2 2nd STAGE (ARRANGED)
D6213 CHANNEL  ; BT/R 2nd STAGE (ARRANGED)
D6220 CHANNEL  ; STAGE DATA
D6500 CHANNEL  ; START INDEX MEMORY
D6502 CHANNEL  ; INDEX MEMORY PARAMETER
D6510 CHANNEL  ; MODEL USED
D6520 CHANNEL  ; PLUG RELIEF SIDE USED
D6521 CHANNEL  ; FRANGE HAVE
D6522 CHANNEL  ; PLUG TYPE
D6523 CHANNEL  ; TIGHT.PRO.No.SELECT
D6524 CHANNEL  ; LOOSEN PRO.No.SELECT
D6600 CHANNEL  ; MODEL NO.(PAGE 31)
D6610 CHANNEL  ; MODEL NAME(PAGE31)
D6620 CHANNEL  ; PLUG RELIEF SIDE
D6623 CHANNEL  ; PROGRAM N/R EDIT RUN WORK NUMBER
D6630 CHANNEL  ; START REGISTER(PAGE31)
D6632 CHANNEL  ; OFFSET REGISTER
D6635 CHANNEL  ; INDEX REGISTER(PAGE31)
D6700 CHANNEL  ; MOUNTH
D6701 CHANNEL  ; :
D6702 CHANNEL  ; DAY
D6703 CHANNEL  ; /2
D6704 CHANNEL  ; 0
D6705 CHANNEL  ; YEAR
D6706 CHANNEL  ; TAB
D6707 CHANNEL  ; HOUR
D6708 CHANNEL  ; :
D6709 CHANNEL  ; MINUTE
D6710 CHANNEL  ; :
D6711 CHANNEL  ; SECOND
D6712 CHANNEL  ; TAB
D6713 CHANNEL  ; LINE No.
D6714 CHANNEL  ; SERIAL No. (6,5 DIGITS)
D6715 CHANNEL  ; SERIAL No. (4,3,2,1 DIGIT)
D6716 CHANNEL  ; SERIAL No. (4,3,2,1 DIGIT)
D6717 CHANNEL  ; TAB
D6718 CHANNEL  ; PART No.(ASCII)
D6719 CHANNEL  ; PART No.(ASCII)
D6720 CHANNEL  ; TAB
D6721 CHANNEL  ; MC No.(ASCII)
D6722 CHANNEL  ; TAB
D6723 CHANNEL  ; TORQUE 1st (XX-.-)
D6724 CHANNEL  ; TORQUE 1st (--X.-)
D6725 CHANNEL  ; TORQUE 1st (---.X)
D6726 CHANNEL  ; ANGLE 1st (XX-.-)
D6727 CHANNEL  ; ANGLE 1st (--X.-)
D6728 CHANNEL  ; ANGLE 1st (---.X)
D6729 CHANNEL  ; SNUG TORQUE 1st (XX-.-)
D6730 CHANNEL  ; SNUG TORQUE 1st (--X.-)
D6731 CHANNEL  ; SNUG TORQUE 1st (---.X)
D6732 CHANNEL  ; TORQUE 2nd (XX-.-)
D6733 CHANNEL  ; TORQUE 2nd (--X.-)
D6734 CHANNEL  ; TORQUE 2nd (---.X)
D6735 CHANNEL  ; ANGLE 2ndXX-.-)
D6736 CHANNEL  ; ANGLE 2nd--X.-)
D6737 CHANNEL  ; ANGLE 2nd (---.X)
D6738 CHANNEL  ; SNUG TORQUE 2nd (XX-.-)
D6739 CHANNEL  ; SNUG TORQUE 2nd (--X.-)
D6740 CHANNEL  ; SNUG TORQUE 2nd (---.X)
D6741 CHANNEL  ; JUDGEMENT(BCD)
D6742 CHANNEL  ; END OF DATA BUFFER
D6800 CHANNEL  ; FIRST WRITE DATA
D6900 CHANNEL  ; MOUNTH (FILENAME)
D6901 CHANNEL  ; DAY (FILENAME)
D6902 CHANNEL  ; YEAR (FILENAME)
D6903 CHANNEL  ; MACHINE No.(FILENAME)
D6904 CHANNEL  ; END OF FILE NAME
D6909 CHANNEL  ; \
D6910 CHANNEL  ; FILENAME WORD 1st
D6914 CHANNEL  ; END OF FILE NAME
D7000 CHANNEL  ; SERIAL No. (XXXX DIGIT)
D7001 CHANNEL  ; LINE No. SERIAL No. (XX XX- - - - DIGIT)
D7002 CHANNEL  ; PART No.
D7003 CHANNEL  ; MC No.
D7004 CHANNEL  ; TORQUE 1st
D7005 CHANNEL  ; ANGLE 1st
D7006 CHANNEL  ; SNUG TORQUE 1st
D7007 CHANNEL  ; TORQUE 2st
D7008 CHANNEL  ; ANGLE 2st
D7009 CHANNEL  ; SNUG TORQUE 2st
D7010 CHANNEL  ; JUDGEMENT
D7200 CHANNEL  ; FIRST SUM. RESULT
D7202 CHANNEL  ; SUM. RESULT LAST
D7500 CHANNEL  ; START INDEX MEMORY
D7502 CHANNEL  ; MODEL OFFSET
D7504 CHANNEL  ; INDEX MEMORY PARAMETER
D7506 CHANNEL  ; MODEL USED
D7508 CHANNEL  ; MODEL SELECTED
D9000 CHANNEL  ; FIRST ID2 DATA READ
D9003 CHANNEL  ; SUM CHECK
D9004 CHANNEL  ; SOUCE FIRST DATA
D9031 CHANNEL  ; FINAL ID_2 DATA READ
D9200 CHANNEL  ; FIRST. CHECK SUM RESUALT ID2
D9202 CHANNEL  ; SUM CHECK
E0_3200.05 BOOL  ; Trigger mc stop
E0_3200.06 BOOL  ; interlock table rotate
E0_3200.09 BOOL  ; PH vacuum blow 1
E0_3200.10 BOOL  ; ph vacuum blow 2
E0_3200.14 BOOL  ; index rotate allowed
E0_3201.06 BOOL  ; safe cond for cyl push product
E0_3201.08 BOOL  ; req disch mode final caulking
E0_3201.10 BOOL  ; out to caulking
E0_3201.11 BOOL  ; PL Diap discharge
E0_3201.14 BOOL  ; to caulking dummy sensor
E0_3300.00 BOOL  ; ITLK.PB FINAL EMERGENCY NOT
E0_3300.01 BOOL  ; ITLK.FINAL CAULKING FUSE CONFIRM
E0_3300.02 BOOL  ; FINAL CAULKING-MASTER ON
E0_3300.03 BOOL  ; ITLK.FINAL CAULKING-ALL HOME
E0_3300.04 BOOL  ; ITLK.FINAL CAULKING DIAPH BLOW OK
E0_3300.05 BOOL  ; ITLK.FINAL CAULKING ABNORMAL DETECTION
E0_3300.06 BOOL  ; disch mode confirm,trigger last work
E0_3300.07 BOOL  ; vacuum 3 OK
E0_3300.08 BOOL  ; ITLK.FINAL CAULKING-AUTO DIAPH VACCUM OK
E0_3300.09 BOOL  ; ITLK.FINAL CAULKING WORK OK
E0_3300.10 BOOL  ; ITLK.FINAL CAULKING WORK OK
E0_3300.11 BOOL  ; ITLK.FINAL CAULKING OPEARTE
E0_3300.12 BOOL  ; ITLK.PH FINAL CAULKING ST1 DETECT
E0_3300.13 BOOL  ; ITLK.PH FINAL CAULKING ST2 DETECT
E0_3300.14 BOOL  ; PH conveyor
E0_3300.15 BOOL  ; table rotate req
E0_3301.00 BOOL  ; Float sensor
E0_3301.01 BOOL  ; Index table in position
E0_3301.02 BOOL  ; lock fwd
E0_3301.03 BOOL  ; absodex ready status
E0_3301.04 BOOL  ; index start coil
E0_3301.06 BOOL  ; Loading OK PL
E0_3301.07 BOOL  ; vacuum start
E0_3301.09 BOOL  ; vacum 1 start
E0_3301.10 BOOL  ; diaph autorun
E0_3301.11 BOOL  ; PB disch mc diap caulking
E0_3301.13 BOOL  ; dummy in feed area
E0_3301.14 BOOL  ; CV RUN
H0.00 BOOL  ; DIAPH BLOW OK
H0.01 BOOL  ; DIAPH VACCUM OK
H0.02 BOOL  ; MB VACCUM OK
H1 CHANNEL  ; MB Loader HaveWork
H100 CHANNEL  ; WorkDiscarg
H12 CHANNEL  ; MB Rotate HaveWork
H12.00 BOOL  ; Vacum work memory
H12.01 BOOL  ; MB Vacuum area
H13 CHANNEL  ; MB ROTATE : FINISH
H13.00 BOOL  ; MB ROTATE : FINISH
H1.00 BOOL  ; MB LOADER : LOADER 1
H1.01 BOOL  ; MB LOADER : LOADER 2
H2 CHANNEL  ; MB Buffer HaveWork
H22 CHANNEL  ; Work Transfer Slide : HAVE Work
H22.00 BOOL  ; TRANSFER SLIDE : HaveWork 1
H22.01 BOOL  ; Work Transfer : BUFFER 2(Stack)
H2.00 BOOL  ; MB LOAD  Positioning area
H300 CHANNEL  ; Oil Apply Auto Sequence
H300.00 BOOL  ; Safe Confirm
H300.01 BOOL  ; Advance & Up Command
H300.02 BOOL  ; Advance, Down Command, & Safe Confirm
H300.03 BOOL  ; Advance, Up Command, & Safe Confirm
H300.04 BOOL  ; Up, Return Command
H300.05 BOOL  ; -
H300.06 BOOL  ; -
H300.07 BOOL  ; -
H300.08 BOOL  ; -
H300.09 BOOL  ; -
H300.10 BOOL  ; -
H300.11 BOOL  ; -
H300.12 BOOL  ; -
H300.13 BOOL  ; -
H300.14 BOOL  ; End Motion
H300.15 BOOL  ; End Cycle
H32 CHANNEL  ; DIAPHAM FEED IN : HAVE WORK
H32.00 BOOL  ; DIAPHAM FEED IN : Buffer1
H400.00 BOOL  ; 001_EMERGENCY STOP
H400.01 BOOL  ; 002_FUSE ABNORMAL
H400.02 BOOL  ; 003_SAFETY COVER OPEN
H400.03 BOOL  ; 004_AIR SOURCE LOW
H400.04 BOOL  ; 005_DEVICE-NET FAULT
H400.05 BOOL  ; 006_PLC ABNORMAL
H400.09 BOOL  ; 010_AIR SOURCE PS. FAULT
H400.10 BOOL  ; 011_DUMMY DOOR OPEN
H400.11 BOOL  ; 012_SHUTTER DOOR INTERRUPTED
H400.12 BOOL  ; 013_FNCK EMERGENCY STOP
H400.13 BOOL  ; 014_FNCK FUSE ABNORMAL
H400.14 BOOL  ; 015_1EC1 ABNORMAL
H400.15 BOOL  ; 016_1EC2 ABNORMAL
H401.00 BOOL  ; 17_1EC3 ABNORMAL
H401.01 BOOL  ; 018_1EC4 ABNORMAL
H401.02 BOOL  ; 19_1MTD1 ABNORMAL
H402.00 BOOL  ; 033_CYCLE TIME OVER
H402.01 BOOL  ; 034_FNCK MASTER OR AUTO STOP
H402.02 BOOL  ; 035_FNCK FAULT OCCER
H402.03 BOOL  ; 036_MB LOADER 1 WORK LOST
H402.04 BOOL  ; 037_MB LOADER 2 WORK LOST
H402.05 BOOL  ; 038_ROTATE UNIT WORK LOST
H402.06 BOOL  ; 039_TRANFER SLIDE MB LOST
H402.07 BOOL  ; 040_DIAPHAM LOADER 1 LOST WORK
H402.08 BOOL  ; 041_DIAPHAM LOADER 2 LOST WORK
H402.09 BOOL  ; 042_DIAPHAM LOADER 3 LOST WORK
H402.10 BOOL  ; 043_DIAPHAM VACCUM STATION WORK LOST
H402.11 BOOL  ; 044_DIAPHAM BUFFER STATION WORK LOST
H402.12 BOOL  ; 045_DIAPHAM FEED IN STATION ABNORMAL
H402.13 BOOL  ; 046_TRANFER SLIDE DIAPHAM LOST
H402.14 BOOL  ; 047_ROTARY GRIPPER 1 LOST WORK
H402.15 BOOL  ; 048_ROTARY GRIPPER 2 LOST WORK
H403.00 BOOL  ; 049_WORK DISCHARGE UNIT WORK LOST
H404.00 BOOL  ; 065_PRODUCTION QUANTITY UP
H404.01 BOOL  ; 066_DEFECT QUANTITY UP
H404.02 BOOL  ; 067_TOTAL QUANTITY UP
H404.03 BOOL  ; 068_ MB LOADER UNIT TIME OVER
H404.04 BOOL  ; 069_MB POSITIONNING UNIT TIME OVER
H404.05 BOOL  ; 070_DIAPHAM FEED IN UNIT TIME OVER
H404.06 BOOL  ; 071_DIAPHAM LOADER UNIT TIME OVER
H404.07 BOOL  ; 072_WORK TRANSFER UNIT TIME OVER
H404.08 BOOL  ; 073_GRIPPER ROTARY UNIT TRANSFER TIME OVER
H404.09 BOOL  ; 074_OK/DISCHARGE UNIT TRANSFER TIME OVER
H405.00 BOOL  ; 81_AS.SHUTTER 1 FAULT
H405.01 BOOL  ; 82_AS.SHUTTER 2 FAULT
H405.02 BOOL  ; 83_AS.DIAPH GRIPPER UNIT FAULT
H405.03 BOOL  ; 84_AS.DIAPH GRIPPER 1 FAULT
H405.04 BOOL  ; 85_AS.DIAPH GRIPPER 2 FAULT
H405.05 BOOL  ; 86_AS.DIAPH GRIPPER 3 FAULT
H405.06 BOOL  ; 87_AS.DIAPH GRIPPER FLIP FAULT
H405.07 BOOL  ; 88_AS.ROTARY GRIPPER 1 FAULT
H405.08 BOOL  ; 89_AS.ROTARY GRIPPER 2 FAULT
H405.09 BOOL  ; 90_AS.ROTARY GRIPPER UNIT 1 FAULT
H405.10 BOOL  ; 91_AS.ROTARY GRIPPER UNIT 2 FAULT
H405.11 BOOL  ; 92_AS.MB LOAD IN FAULT
H405.12 BOOL  ; 93_AS.MB LOAD OUT FAULT
H405.13 BOOL  ; 94_AS.MB LOAD OUT UNIT FAULT
H405.14 BOOL  ; 95_AS.MB SLIDE UNIT FAULT
H405.15 BOOL  ; 96_AS.MB POSITION PIN UNIT FAULT
H406.00 BOOL  ; 97_AS.WORK TRANSFER UNIT FAULT
H406.01 BOOL  ; 098_AS.FINISH TRAY FAULT
H406.02 BOOL  ; 099_AS.OK PUSH FAULT
H406.03 BOOL  ; 100_AS.NG PULL FAULT
H406.04 BOOL  ; NG BOX FULL
H406.05 BOOL  ; 102_WORK FINISH FULL
H406.06 BOOL  ; 103_SAFET DOOR IS OPEN
H406.07 BOOL  ; 104_
H406.08 BOOL  ; 105_
H406.09 BOOL  ; 106_
H406.10 BOOL  ; 107_FASTENING TRQ HIGH NG
H406.11 BOOL  ; 108_FASTENING TRQ LOW NG
H406.12 BOOL  ; 109_FASTENING ANG HIGH NG
H406.13 BOOL  ; 110_FASTENING ANG LOW NG
H406.14 BOOL  ; 111_FASTENING TIME MIN NG
H406.15 BOOL  ; 112_FASTENING TIME MAX NG
H407.00 BOOL  ; 113_FASTENING MON. TRQ HIGH NG
H407.01 BOOL  ; 114_FASTENING MON. TRQ LOW NG
H407.02 BOOL  ; 115_FASTENING T/R1 HIGH NG
H407.03 BOOL  ; 116_FASTENING T/R1 LOW NG
H407.04 BOOL  ; 117_FASTENING T/R2 HIGH NG
H407.05 BOOL  ; 118_FASTENING T/R2 LOW NG
H407.06 BOOL  ; 119_FASTENING BT/R HIGH NG
H407.07 BOOL  ; 120_FASTENING B/TR LOW NG
H407.08 BOOL  ; 121_P/N DOES NOT MATCH
H407.09 BOOL  ; 122_ID WRITE ERROR
H407.10 BOOL  ; 123_PALLATE NG.FULL
H408.13 BOOL  ; 125_FIotNotReady
H408.14 BOOL  ; 126_FIotQtyInfoHS1Ans.Fault
H408.15 BOOL  ; 127_FIoT Disable
H41 CHANNEL  ; DPH Loader Have work
H410.00 BOOL  ; 161_PRODUCTION QUANTITY WARNING
H410.01 BOOL  ; 162_DEFECT QUANTITY WARNING
H410.02 BOOL  ; 163_TOTAL QUANTITY WARNING
H410.03 BOOL  ; 164_CT4 COUNTING WARNING
H410.04 BOOL  ; 165_CT5 COUNTING WARNING
H410.05 BOOL  ; 166_CT6 COUNTING WARNING
H410.06 BOOL  ; 167_CT7 COUNTING WARNING
H410.07 BOOL  ; 168_CT8 COUNTING WARNING
H410.08 BOOL  ; 169_
H410.09 BOOL  ; 170_WIP DISCHARGE DONE
H410.10 BOOL  ; 171_TIGHTEN SLIDE 1 TIGHT TIM OVER
H410.11 BOOL  ; 172_TIGHTEN SLIDE 1 HOME TIM OVER
H410.12 BOOL  ; 173_TIGHTEN SLIDE 2 RET. TIM OVER
H410.13 BOOL  ; 174_TIGHTEN SLIDE 2 ADV. TIM OVER
H410.14 BOOL  ; 175_WORK CLMP. 1 DOWN TIM OVER
H410.15 BOOL  ; 176_WORK CLMP. 1 UP TIM OVER
H411.00 BOOL  ; 177_WORK CLMP. 2 DOWN TIM OVER
H411.01 BOOL  ; 178_WORK CLMP. 2 UP TIM OVER
H411.02 BOOL  ; 179_WORK CLMP. 3 PRESS CLAMP 1 TIM OVER
H411.03 BOOL  ; 180_WORK CLMP. 3 PRESS CLAMP 2 TIM OVER
H411.04 BOOL  ; 181_WORK CLMP. 3 NOT PRESS CLAMP TIM OVER
H411.05 BOOL  ; 182_DUMMY FRANGE 1 CLAMP TIM OVER
H411.06 BOOL  ; 183_DUMMY FRANGE 1 NOT CLAMP TIM OVER
H411.07 BOOL  ; 184_DUMMY FRANGE 2 CLAMP TIM OVER
H411.08 BOOL  ; 185_DUMMY FRANGE 2 NOT CLAMP TIM OVER
H411.09 BOOL  ; 186_JIG CHANGE OVER MIRROR TIM OVER
H411.10 BOOL  ; 187_JIG CHANGE OVER NORMAL TIM OVER
H411.11 BOOL  ; 188_NUT RUNNER CHG.OVER MIRROR TIM OVER
H411.12 BOOL  ; 189_NUT RUNNER CHG.OVER NORMAL TIM OVER
H411.13 BOOL  ; 190_WORK CLAMP CHG.OVER MIRROR TIM OVER
H411.14 BOOL  ; 191_WORK CLAMP CHG.OVER NORMAL TIM OVER
H411.15 BOOL  ; 192_SAFETY COVER CLOSE TIM OVER
H412.00 BOOL  ; 193_SAFETY COVER OPEN TIM OVER
H412.01 BOOL  ; 194_WORK CLMP. 1 DOWN FRANGE TIM OVER
H412.02 BOOL  ; 195_WORK CLMP. 2 DOWN FRANGE TIM OVER
H412.03 BOOL  ; 196_
H412.04 BOOL  ; 197_
H412.05 BOOL  ; 198_
H412.06 BOOL  ; 199_
H412.07 BOOL  ; 200_PLC LOW BATTERY
H412.08 BOOL  ; 201_MU LOW BATTERY
H412.09 BOOL  ; 202_AU LOW BATTERY
H415.01 BOOL  ; EMERGENCY STOP ALL
H415.02 BOOL  ; AUTO STOP FAULT
H415.03 BOOL  ; CYCLE STOP
H415.04 BOOL  ; FAULT STOP ALL
H415.05 BOOL  ; WARNING
H415.07 BOOL  ; FAULT MOTION
H415.15 BOOL  ; ALL FAULT(OFF)
H416.00 BOOL  ; AL FAULT(OFF) TOWER LAMP
H41.00 BOOL  ; DIAPH LOADER : LOADER STATUS1
H41.01 BOOL  ; DIAPH LOADER : LOADER STATUS2
H41.02 BOOL  ; DIAPH LOADER : LOADER STATUS3
H42 CHANNEL  ; DPH Load buffer Have work
H420.00 BOOL  ; ASSIST11-1
H420.01 BOOL  ; ASSIST11-2
H420.02 BOOL  ; ASSIST11-3
H420.03 BOOL  ; ASSIST11-4
H420.04 BOOL  ; ASSIST11-5
H420.05 BOOL  ; ASSIST11-6
H420.06 BOOL  ; ASSIST11-7
H420.07 BOOL  ; ASSIST11-8
H420.08 BOOL  ; ASSIST12-1
H420.09 BOOL  ; ASSIST12-2
H420.10 BOOL  ; ASSIST12-3
H420.11 BOOL  ; ASSIST12-4
H420.12 BOOL  ; ASSIST12-5
H420.13 BOOL  ; ASSIST12-6
H420.14 BOOL  ; ASSIST12-7
H420.15 BOOL  ; ASSIST12-8
H424.00 BOOL  ; ASSIST21-1
H424.01 BOOL  ; ASSIST21-2
H424.02 BOOL  ; ASSIST21-3
H424.03 BOOL  ; ASSIST21-4
H424.04 BOOL  ; ASSIST21-5
H424.05 BOOL  ; ASSIST21-6
H424.06 BOOL  ; ASSIST21-7
H424.07 BOOL  ; ASSIST21-8
H424.08 BOOL  ; ASSIST22-1
H424.09 BOOL  ; ASSIST22-2
H424.10 BOOL  ; ASSIST22-3
H424.11 BOOL  ; ASSIST22-4
H424.12 BOOL  ; ASSIST22-5
H424.13 BOOL  ; ASSIST22-6
H424.14 BOOL  ; ASSIST22-7
H424.15 BOOL  ; ASSIST22-8
H428.00 BOOL  ; ASSIST31-1
H428.01 BOOL  ; ASSIST31-2
H428.02 BOOL  ; ASSIST31-3
H428.03 BOOL  ; ASSIST31-4
H428.04 BOOL  ; ASSIST31-5
H428.05 BOOL  ; ASSIST31-6
H428.06 BOOL  ; ASSIST31-7
H428.07 BOOL  ; ASSIST31-8
H428.08 BOOL  ; ASSIST32-1
H428.09 BOOL  ; ASSIST32-2
H428.10 BOOL  ; ASSIST32-3
H428.11 BOOL  ; ASSIST32-4
H428.12 BOOL  ; ASSIST32-5
H428.13 BOOL  ; ASSIST32-6
H428.14 BOOL  ; ASSIST32-7
H428.15 BOOL  ; ASSIST32-8
H42.00 BOOL  ; DIAPH BUFFER : VACCUM STATUS1
H42.01 BOOL  ; DIAPH BUFFER : BUFFER STATUS2
H432.00 BOOL  ; ASSIST41-1
H432.01 BOOL  ; ASSIST41-2
H432.02 BOOL  ; ASSIST41-3
H432.03 BOOL  ; ASSIST41-4
H432.04 BOOL  ; ASSIST41-5
H432.05 BOOL  ; ASSIST41-6
H432.06 BOOL  ; ASSIST41-7
H432.07 BOOL  ; ASSIST41-8
H432.08 BOOL  ; ASSIST42-1
H432.09 BOOL  ; ASSIST42-2
H432.10 BOOL  ; ASSIST42-3
H432.11 BOOL  ; ASSIST42-4
H432.12 BOOL  ; ASSIST42-5
H432.13 BOOL  ; ASSIST42-6
H432.14 BOOL  ; ASSIST42-7
H432.15 BOOL  ; ASSIST42-8
H436.00 BOOL  ; ASSIST51-1
H436.01 BOOL  ; ASSIST51-2
H436.02 BOOL  ; ASSIST51-3
H436.03 BOOL  ; ASSIST51-4
H436.04 BOOL  ; ASSIST51-5
H436.05 BOOL  ; ASSIST51-6
H436.06 BOOL  ; ASSIST51-7
H436.07 BOOL  ; ASSIST51-8
H436.08 BOOL  ; ASSIST52-1
H436.09 BOOL  ; ASSIST52-2
H436.10 BOOL  ; ASSIST52-3
H436.11 BOOL  ; ASSIST52-4
H436.12 BOOL  ; ASSIST52-5
H436.13 BOOL  ; ASSIST52-6
H436.14 BOOL  ; ASSIST52-7
H436.15 BOOL  ; ASSIST52-8
H440.00 BOOL  ; ASSIST61-1
H440.01 BOOL  ; ASSIST61-2
H440.02 BOOL  ; ASSIST61-3
H440.03 BOOL  ; ASSIST61-4
H440.04 BOOL  ; ASSIST61-5
H440.05 BOOL  ; ASSIST61-6
H440.06 BOOL  ; ASSIST61-7
H440.07 BOOL  ; ASSIST61-8
H440.08 BOOL  ; ASSIST62-1
H440.09 BOOL  ; ASSIST62-2
H440.10 BOOL  ; ASSIST62-3
H440.11 BOOL  ; ASSIST62-4
H440.12 BOOL  ; ASSIST62-5
H440.13 BOOL  ; ASSIST62-6
H440.14 BOOL  ; ASSIST62-7
H440.15 BOOL  ; ASSIST62-8
H444.00 BOOL  ; ASSIST71-1
H444.01 BOOL  ; ASSIST71-2
H444.02 BOOL  ; ASSIST71-3
H444.03 BOOL  ; ASSIST71-4
H444.04 BOOL  ; ASSIST71-5
H444.05 BOOL  ; ASSIST71-6
H444.06 BOOL  ; ASSIST71-7
H444.07 BOOL  ; ASSIST71-8
H444.08 BOOL  ; ASSIST72-1
H444.09 BOOL  ; ASSIST72-2
H444.10 BOOL  ; ASSIST72-3
H444.11 BOOL  ; ASSIST72-4
H444.12 BOOL  ; ASSIST72-5
H444.13 BOOL  ; ASSIST72-6
H444.14 BOOL  ; ASSIST72-7
H444.15 BOOL  ; ASSIST72-8
H51 CHANNEL  ; RotaryGP1 HAVE WORK
H51.00 BOOL  ; ROTARY GRIP 1 : LOADER 1
H58 CHANNEL  ; RotaryGP1 OK-NG
H61 CHANNEL  ; RotaryGripper2 HAVE WORK
H61.00 BOOL  ; ROTARY GRIP 2 : LOADER 1
H62 CHANNEL  ; RotaryGP2 : HAVE WorK
H63 CHANNEL  ; RotaryGrip2 : STATUS
H68 CHANNEL  ; RotaryGP2 [OK=1,NG=2]
H72 CHANNEL  ; Work Discharge : Have Work
H72.00 BOOL  ; WORK DISCHARGE : Have work
H73 CHANNEL  ; OK/NG Discharge : Status
H78 CHANNEL  ; WORK DISCHARGE : OK/NG
H82 CHANNEL  ; FinalCualking ST1 HaveWork (1:have work 2:no work)
H82.00 BOOL  ; FINAL CAULKING ST1 DETECT MEM Have work
H82.01 BOOL  ; FINAL CAULKING ST1 : Not have work
H82.02 BOOL  ; FINAL CAULKING ST1 DETECT MEM
H83 CHANNEL  ; FNCK Rotary Table Operate
H88 CHANNEL  ; FinalCualking ST1 Judge [OK=1,NG=2]
H88.00 BOOL  ; FINAL CAULKING ST1 RESULT OK
H88.01 BOOL  ; FINAL CAULKING ST1 RESULT NG
H92 CHANNEL  ; FinalCualking ST2 HaveWork
H92.00 BOOL  ; FINAL CAULKING ST2 DETECT MEM Have work
H92.01 BOOL  ; FINAL CAULKING ST2 : Not have work
H99.00 BOOL  ; RotaryGripperInterlock
T0000 BOOL  ; START UP
T0001 BOOL  ; SAFETY COVER CLOSE DELAY
T0020 BOOL  ; Oil Apply Auto Trigger Delay
T0035 BOOL  ; DELAY CF DAT SENT
T0050 BOOL  ; ABORT START
T0056 BOOL  ; TIMER
T0057 BOOL  ; TIMER
T0058 BOOL  ; TIMER
T0059 BOOL  ; TIMER
T0060 BOOL  ; TIMER
T0061 BOOL  ; TIMER
T0062 BOOL  ; TIMER
T0064 BOOL  ; TIMER
T0079 BOOL  ; FOR DELAY LATCH W260.05
T0087 BOOL  ; ADD SOUND FAULT ID2
T0088 BOOL  ; ADD SOUND TIME 3 SEC
T0089 BOOL  ; DELAY CONF. EN/DIS
T0100 BOOL  ; PB.EMER STOP
T0101 BOOL  ; AIR SOURCE CONFIRM.
T0102 BOOL  ; AUTO.IND.(AUTO=on)
T0103 BOOL  ; PB.MASTER ON
T0104 BOOL  ; PB.AUTO RUN
T0105 BOOL  ; PB.CYCLE STOP
T0106 BOOL  ; PB.DUMMY DOOR OPEN REQUEST
T0107 BOOL  ; CR.TEACHING ON
T0108 BOOL  ; CR.MACHINR DOOR CONFIRM
T0109 BOOL  ; CR.DUMMY DOOR CONFIRM
T0110 BOOL  ; CR.SHUTTER DOOR OUT CONFIRM
T0111 BOOL  ; CR.SHUTTER DOOR IN CONFIRM
T0112 BOOL  ; CR.MASTER ON CONFIRM
T0113 BOOL  ; CR.FUSE NORMAL CONFIRM
T0114 BOOL  ; CR.DIAPHAM DOOR ENABLE CONF
T0115 BOOL  ; .
T0116 BOOL  ; P3SH MASTER OK DELAY
T0117 BOOL  ; P3SH MASTER NG DELAY
T0120 BOOL  ; DELAY TIME
T0130 BOOL  ; DELAY FAULT SOL.ASSY
T0162 BOOL  ; DELAY SENSER CLEAR PICKKING ABNORMAL
T0170 BOOL  ; CYCLE TIME OVER
T0171 BOOL  ; DELAY DATA FROM ID FINISH
T0173 BOOL  ; TIME TO RESET DATA
T0174 BOOL  ; BUZZER TIMMER
T0175 BOOL  ; CYCLE TIME CONTROL ROTATE
T0176 BOOL  ; PLUG OIL SUPPLY CONF.
T0186 BOOL  ; CHECK PLUG MODEL DELAY TIME
T0190 BOOL  ; DELAY CONF.
T0200 BOOL  ; ITLK.PB FINAL EMERGENCY NOT
T0201 BOOL  ; ITLK.FINAL CAULKING FUSE CONFIRM
T0202 BOOL  ; ITLK.FINAL CAULKING-MASTER ON
T0203 BOOL  ; ITLK.FINAL CAULKING-ALL HOME
T0204 BOOL  ; ITLK.FINAL CAULKING-AUTO RUNNING
T0205 BOOL  ; ITLK.FINAL CAULKING ABNORMAL DETECTION
T0207 BOOL  ; ITLK.FINAL CAULKING-AUTO M&B VACCUM OK
T0208 BOOL  ; ITLK.FINAL CAULKING-AUTO DIAPH VACCUM OK
T0209 BOOL  ; ITLK.FINAL CAULKING WORK OK
T0210 BOOL  ; ITLK.FINAL CAULKING WORK NG
T0211 BOOL  ; ITLK.FINAL CAULKING WORK FINISH
T0212 BOOL  ; ITLK.PH FINAL CAULKING ST1 DETECT
T0213 BOOL  ; ITLK.PH FINAL CAULKING ST2 DETECT
T0251 BOOL  ; PH. DUMMY FEED IN CONFIRM
T0252 BOOL  ; PH. WORK FULL
T0253 BOOL  ; PH.TRANSFER STATION DIAPH SIDE CONFIRM
T0254 BOOL  ; PH.TRANSFER STATION DIAPH WORK CONFIRM
T0255 BOOL  ; PH.TRANSFER STATION M&B WORK CONFIRM
T0256 BOOL  ; PH. M&B LOADER WORK CONF 1
T0257 BOOL  ; PH. M&B LOADER WORK CONF 2
T0258 BOOL  ; PH. WORK IN ROTATE UNIT CONFIRM
T0259 BOOL  ; PH. WORK M&B FEED IN CONFIRM
T0260 BOOL  ; PH. WORK ROTATE PRE-END CONFIRM
T0261 BOOL  ; PH. TEMINAL IN POSITION CONFIRM
T0262 BOOL  ; PH. WORK DIAPH LOAD IN CONFIRM
T0263 BOOL  ; PH.STATION DIAPH VACCUM CONFIRM
T0264 BOOL  ; PH.STATION BUFFER DIAPH CONFIRM
T0265 BOOL  ; PH. WORK NG CONFIRM
T0266 BOOL  ; PH. WORK OK CONFIRM
T0289 BOOL  ; DELAY CHECK SCAN TIME MEMORY
T0290 BOOL  ; DELAY CHECK MU BATTERY
T0291 BOOL  ; DELAY CHECK AU BATTERY
T0300 BOOL  ; PRESSURE CONF. on [CR.001]
T0301 BOOL  ; PRESSURE CONF. off [CR.001]
T0302 BOOL  ; MASTER ON CONF. on[CR.002]
T0303 BOOL  ; MASTER ON CONF. off[CR.002]
T0304 BOOL  ; SAFETY.SLIDE CONF. on [CR.003]
T0305 BOOL  ; SAFETY.SLIDE CONF. off [CR.003]
T0306 BOOL  ; SAFETY.COV.1 CLOSE CONF. on [CR.004]
T0307 BOOL  ; SAFETY.COV.1 CLOSE CONF. off [CR.004]
T0308 BOOL  ; AUTO MODE [SS.005]
T0309 BOOL  ; IND. MODE [SS.005]
T0310 BOOL  ; SPEED CONTRL. ALRM. on [CR.006]
T0311 BOOL  ; SPEED CONTRL. ALRM. off [CR.006]
T0312 BOOL  ; FUSE OK on [CR.007]
T0313 BOOL  ; FUSE OK off [CR.007]
T0314 BOOL  ; WORK CLMP.3 PRESS CLMP.1 on [PX.206]
T0315 BOOL  ; WORK CLMP.3 PRESS CLMP.1 off [PX.206]
T0316 BOOL  ; WORK CLMP.3 PRESS CLMP.2 on [PX.207]
T0317 BOOL  ; WORK CLMP.3 PRESS CLMP.2 off [PX.207]
T0318 BOOL  ; NG WORK CONF. on [PH.208]
T0319 BOOL  ; NG WORK CONF. off [PH.208]
T0320 BOOL  ; MGH1 CUT OFF1
T0321 BOOL  ; MGH1 CUT OFF2
T0322 BOOL  ; MGH2 CUT OFF1
T0323 BOOL  ; MGH2 CUT OFF2
T0324 BOOL  ; SOCKET CONF. SENSOR 2 on [PH.212]
T0325 BOOL  ; SOCKET CONF. SENSOR 2 off [PH.212]
T0326 BOOL  ; SOCKET CONF. SENSOR 3 on [PH.213]
T0327 BOOL  ; SOCKET CONF. SENSOR 3 off [PH.213]
T0328 BOOL  ; PLUG CONF. on [PH.214]
T0329 BOOL  ; PLUG CONF. off [PH.214]
T0330 BOOL  ; WORK CONF. on[PH.215]
T0331 BOOL  ; WORK CONF. off[PH.215]
T0332 BOOL  ; DELAY CONF.
T0334 BOOL  ; DELAY AS.ADD
T0335 BOOL  ; DELAY AS.ADD
T0336 BOOL  ; DELAY TIME
T0337 BOOL  ; DELAY TIME
T0338 BOOL  ; DELAY TIME
T0339 BOOL  ; DELAY TIME
T0340 BOOL  ; DELAY TIME
T0341 BOOL  ; DELAY TIME
T0342 BOOL  ; DELAY TIME
T0343 BOOL  ; DELAY TIME
T0344 BOOL  ; DELAY TIME
T0345 BOOL  ; DELAY TIME
T0346 BOOL  ; DELAY TIME
T0347 BOOL  ; DELAY TIME
T0351 BOOL  ; PH. DUMMY FEED IN CONFIRM off
T0352 BOOL  ; PH. WORK FULL off
T0353 BOOL  ; PH.TRANSFER STATION DIAPH SIDE CONFIRM off
T0354 BOOL  ; PH.TRANSFER STATION DIAPH WORK CONFIRM off
T0355 BOOL  ; PH.TRANSFER STATION M&B WORK CONFIRM off
T0356 BOOL  ; PH. M&B LOADER WORK CONF 1 off
T0357 BOOL  ; PH. M&B LOADER WORK CONF 2 off
T0358 BOOL  ; PH. WORK IN ROTATE UNIT CONFIRM off
T0359 BOOL  ; PH. WORK M&B FEED IN CONFIRM off
T0360 BOOL  ; PH. WORK ROTATE PRE-END CONFIRM off
T0361 BOOL  ; PH. TEMINAL IN POSITION CONFIRM off
T0362 BOOL  ; PH. WORK DIAPH LOAD IN CONFIRM off
T0363 BOOL  ; PH.STATION DIAPH VACCUM CONFIRM off
T0364 BOOL  ; PH.STATION BUFFER DIAPH CONFIRM off
T0365 BOOL  ; PH. WORK NG CONFIRM off
T0366 BOOL  ; PH. WORK OK CONFIRM off
T0400 BOOL  ; Delay time
T0410 BOOL  ; Delay
T0431 BOOL  ; MANUAL ON
T0432 BOOL  ; OUTPUT 1 LOW ENERGY 1 MINUTE CLOCK
T0433 BOOL  ; OUTPUT 2 LOW ENERGY 1 MINUTE CLOCK
T0434 BOOL  ; OUTPUT 3 LOW ENERGY 1 MINUTE CLOCK
T0435 BOOL  ; OUTPUT 4 LOW ENERGY 1 MINUTE CLOCK
T0436 BOOL  ; OUTPUT 5 LOW ENERGY 1 MINUTE CLOCK
T0437 BOOL  ; OUTPUT 1 START DELAY 1 MINUTE CLOCK
T0438 BOOL  ; OUTPUT 2 START DELAY 1 MINUTE CLOCK
T0439 BOOL  ; OUTPUT 3 START DELAY 1 MINUTE CLOCK
T0440 BOOL  ; OUTPUT 4 START DELAY 1 MINUTE CLOCK
T0441 BOOL  ; OUTPUT 5 START DELAY 1 MINUTE CLOCK
T0442 BOOL  ; OUTPUT 1 BREAK DELAY 1 MINUTE CLOCK
T0443 BOOL  ; OUTPUT 2 BREAK DELAY 1 MINUTE CLOCK
T0444 BOOL  ; OUTPUT 3 BREAK DELAY 1 MINUTE CLOCK
T0445 BOOL  ; OUTPUT 4 BREAK DELAY 1 MINUTE CLOCK
T0446 BOOL  ; OUTPUT 5 BREAK DELAY 1 MINUTE CLOCK
T0450 BOOL  ; POWER ON TIMER
T0471 BOOL  ; WATCH_DOG_TIMER
T0506 BOOL  ; .
T0515 BOOL  ; DELAY CONF. STARTR READ ID2
T0521 BOOL  ; ALMF021_Oil Apply UD Fault
T0522 BOOL  ; ALMF022_Oil Apply AR Fault
T0530 BOOL  ; DELAY PALLATE FULL
T0712 BOOL  ; WAIT PREPARE DATA COMPLETE
T0713 BOOL  ; WAIT PREPARE DATA COMPLETE
T0720 BOOL  ; TIME TO WAIT
T0750 BOOL  ; MB LOAD IN TIMER
T1000 BOOL  ; DELAY AUTO ADD END
T1002 BOOL  ; DELAY FOR RUN N/R P.20
T1050 BOOL  ; DELAY FOR RUN N/R P20 ST1
T1051 BOOL  ; DELAY AUTO END P20
T1060 BOOL  ; DELAY FOR RUN N/R PROGRAM REERUN ST1
T1061 BOOL  ; DELAY AUTO END PROGRAM REERUN
T1070 BOOL  ; DELAY CONF. DATA CHECK TRQ
T1100 BOOL  ; DELAY AUTO ADD P21 END
T1102 BOOL  ; DELAY FOR RUN N/R P.21
T1606 BOOL  ; CHUCK CONf
T1629 BOOL  ; CHUCK CONF
T1630 BOOL  ; CHUCK CONF
T1657 BOOL  ; CHUCK CONF
T1659 BOOL  ; CHUCK CONF
T1661 BOOL  ; CHUCK CONF
T1690 BOOL  ; CHUCK CONF
T1715 BOOL  ; CHUCK CONF
T1717 BOOL  ; CHUCK CONF
T1801 BOOL  ; Time Delay
T2000 BOOL  ; PB.EMERGENCY STOP CONFIRM on 0.00
T2008 BOOL  ; SOL.GIPPER TRANSFER 1 CHUCK CONF
T2010 BOOL  ; SOL.GIPPER TRANSFER 2 CHUCK CONF
T2012 BOOL  ; SOL.GIPPER TRANSFER 2 UNCHUCK CONF
T2022 BOOL  ; SOL.GIPPER TRANSFER 2 CHUCK CONF
T2069 BOOL  ; SOL.GIPPER TRANSFER 2 CHUCK CONF
T2070 BOOL  ; SOL.GIPPER TRANSFER 1 CHUCK CONF
T2071 BOOL  ; SOL.GIPPER TRANSFER 2 CHUCK CONF
T2072 BOOL  ; SOL.GIPPER TRANSFER 2 CHUCK CONF
T2079 BOOL  ; SOL.GIPPER TRANSFER 2 CHUCK CONF
T2081 BOOL  ; SOL.GIPPER TRANSFER 1 CHUCK CONF
T2123 BOOL  ; SOL.GIPPER TRANSFER 2 CHUCK CONF
T2408 BOOL  ; GRIPPER 1 DIAPH CHUCK CONF
T2410 BOOL  ; GRIPPER 2 DIAPH CHUCK CONF
T2421 BOOL  ; GRIPPER 1 DIAPH CHUCK CONF
T2432 BOOL  ; GRIPPER 1 DIAPH UNCHUCK CONF
T2434 BOOL  ; GRIPPER 2 DIAPH UNCHUCK CONF
T470 CHANNEL  ; CYCLE TIME MEASUREMENT
T471 CHANNEL  ; WATCH_DOG_TIMER
T506 CHANNEL  ; WAITING-TIME TIMER
W0.00 BOOL  ; PB.NOT EMERGENCY STOP
W100.14 BOOL  ; CR.DIAPHAM DOOR ENABLE CONF
W100.15 BOOL  ; .
W101.00 BOOL  ; ITLK.PB FINAL EMERGENCY NOT
W101.01 BOOL  ; ITLK.FINAL CAULKING FUSE CONFIRM
W101.02 BOOL  ; ITLK.FINAL CAULKING-MASTER ON,AUTO RUNNING
W101.03 BOOL  ; ITLK.FINAL CAULKING-ALL HOME
W101.04 BOOL  ; vacuum blow 2 ok
W101.05 BOOL  ; ITLK.FINAL CAULKING ABNORMAL DETECTION
W101.06 BOOL  ; .
W101.07 BOOL  ; vacuum blow 3 start
W101.08 BOOL  ; VACUUM Blow 1 OK
W101.09 BOOL  ; ITLK.FINAL CAULKING WORK OK
W101.10 BOOL  ; ITLK.FINAL CAULKING WORK NG
W101.11 BOOL  ; ITLK.FINAL CAULKING OPEARTE
W101.12 BOOL  ; ITLK.PH FINAL CAULKING ST1 DETECT
W101.13 BOOL  ; ITLK.PH FINAL CAULKING ST2 DETECT
W101.14 BOOL  ; .
W101.15 BOOL  ; .
W102.08 BOOL  ; 1EC3.MIDDLE COMPLETE
W102.13 BOOL  ; .
W102.14 BOOL  ; .
W102.15 BOOL  ; .
W107.03 BOOL  ; PROHIBIT MOVE
W10.00 BOOL  ; COIL ADJ. SPARE1
W10.01 BOOL  ; COIL ADJ. SPARE2
W10.02 BOOL  ; COIL ADJ. SPARE3
W10.03 BOOL  ; COIL ADJ. SPARE4
W10.04 BOOL  ; COIL ADJ. SPARE5
W10.05 BOOL  ; COIL ADJ. SPARE6
W10.06 BOOL  ; COIL ADJ. SPARE7
W10.07 BOOL  ; COIL ADJ. SPARE8
W110.00 BOOL  ; MASTER CHECK CONDITION
W110.01 BOOL  ; MASTER CHECK START
W110.02 BOOL  ; MASTER GD-P3S CONFIRM on
W110.03 BOOL  ; MASTER GD-P3S CONFIRM off
W110.04 BOOL  ; MASTER GD-P3SH CONFIRM on
W110.05 BOOL  ; MASTER GD-P3SH CONFIRM off
W110.15 BOOL  ; GD-P3S MASTER OK
W111.00 BOOL  ; P3S MASTER CHECK CONDITION
W111.01 BOOL  ; PUSHER DOWN
W111.02 BOOL  ; PUSHER DOWN CONFIRM
W111.03 BOOL  ; GD-P3S MASTER OK
W111.04 BOOL  ; GD-P3S MASTER NG
W111.05 BOOL  ; GD-P3S MASTER CHECK OK
W111.06 BOOL  ; WORK PUSHER UP
W111.07 BOOL  ; WORK PUSHER UP CONFIRM
W111.15 BOOL  ; P3S MASTER CHECK COMPLETE
W112.00 BOOL  ; P3SH MASTER CHECK CONDITION
W112.01 BOOL  ; PUSHER DOWN
W112.02 BOOL  ; PUSHER DOWN CONFIRM
W112.03 BOOL  ; GD-P3SH MASTER OK
W112.04 BOOL  ; GD-P3SH MASTER NG
W112.05 BOOL  ; GD-P3SH MASTER CHECK OK
W112.06 BOOL  ; WORK PUSHER UP
W112.07 BOOL  ; WORK PUSHER UP CONFIRM
W112.15 BOOL  ; P3SH MASTER CHECK COMPLETE
W113.03 BOOL  ; GD-P3SH MASTER OK
W120.00 BOOL  ; IND. START TRQ HI
W120.01 BOOL  ; IND. START TRQ MID
W120.02 BOOL  ; IND. START TRQ LOW
W120.03 BOOL  ; IND. START SPEED HI
W120.04 BOOL  ; IND. START SPEED MID
W120.05 BOOL  ; IND. START SPEED LOW
W130.00 BOOL  ; IND. MASTER TEST START TRQ HI.CONF
W130.01 BOOL  ; IND. MASTER TEST START TRQ MID.CONF
W130.02 BOOL  ; IND. MASTER TEST START TRQ LOW.CONF
W130.03 BOOL  ; IND. MASTER TEST START SPEED HI.CONF
W130.04 BOOL  ; IND. MASTER TEST START SPEED MID.CONF
W130.05 BOOL  ; IND. MASTER TEST START SPEED LOW.CONF
W130.15 BOOL  ; START CONF. MASTER CHECK TEST N/R
W152.12 BOOL  ; .
W152.13 BOOL  ; .
W152.14 BOOL  ; .
W152.15 BOOL  ; .
W153.06 BOOL  ; .
W153.15 BOOL  ; .
W154.00 BOOL  ; AS.WORK FINISH TRAY DOWN CONFIRM
W154.01 BOOL  ; AS.WORK FINISH TRAY UP CONFIRM
W154.02 BOOL  ; AS.OK PUSH UP. CONFIRM
W154.03 BOOL  ; AS.OK PUSH DOWN. CONFIRM
W154.04 BOOL  ; AS.NG PUSH DOWN. CONFIRM
W154.05 BOOL  ; AS.NG PUSH UP. CONFIRM
W154.06 BOOL  ; .
W154.07 BOOL  ; PH. WORK M&B FEED IN CONFIRM
W155.07 BOOL  ; PH. MB FEED IN CONFIRM off
W157.00 BOOL  ; STOPPER 1 DOWN CONF.
W157.01 BOOL  ; STOPPER 1 UP CONF.
W199.00 BOOL  ; DISCHARGE PROCESS START
W199.01 BOOL  ; MB DISCHARGE END
W199.02 BOOL  ; MB ROTATE DISCHARGE END
W199.03 BOOL  ; DIAPHAM IN DISHARGE END
W199.04 BOOL  ; DIAPHAM LOADER DISHARGE END
W199.05 BOOL  ; TRANSFER WORK DISHARGE END
W199.06 BOOL  ; ROTARY GRIPPER DISCHARGE END
W199.07 BOOL  ; OK/NG END
W199.14 BOOL  ; DUMMY DOOR ENABLE
W199.15 BOOL  ; WORK DISCHARGE END ALL
W1.00 BOOL  ; PC NORMAL AUX.
W1.01 BOOL  ; PC NORMAL
W1.02 BOOL  ; D-NET UNIT 1:NORMAL
W200.00 BOOL  ; OPERATION PLUG ASSY CONDITION
W200.01 BOOL  ; OPERATION PLUG ASSY CONDITION 1
W200.03 BOOL  ; READ ID_2 TACK
W200.04 BOOL  ; READ ID_2 TACK CONF.
W200.05 BOOL  ; TAKE WORK FORM OIL SPY
W200.06 BOOL  ; AUTO ASSY TAKE WORK OIL SPY CONF
W200.07 BOOL  ; WRITE ID2
W200.08 BOOL  ; AUTO ASSY WRITE ID2 CONF.
W200.09 BOOL  ; AUOT ASSY SOL.ADV.
W200.10 BOOL  ; AUTO PLUG ASSY SOL.ADV. CONF.
W200.11 BOOL  ; CONF.FREM TAKE JIG
W200.12 BOOL  ; CONF.FREM TAKE JIG CONF.
W200.13 BOOL  ; AUTO ASSY PLUG SOL.RTN.
W200.14 BOOL  ; AUTO ASSY PLUG SOL.RTN.CONF
W200.15 BOOL  ; AUTO ASSY PLUG LOOP FINISH
W201.03 BOOL  ; CALL LAMP AREA PICKKING SENSOR
W201.04 BOOL  ; PICK BOLT CF.PLUG ASSY
W201.05 BOOL  ; PLUG ASSY WAIT PICK OIL SPAY
W201.06 BOOL  ; CF.WORK TO OIL SPAY
W202.00 BOOL  ; OPERATION CHANG TRAY
W205.00 BOOL  ; FAULT ADD ID2
W205.05 BOOL  ; BUZZER ID2 ALRAM
W205.06 BOOL  ; BUZZER RESET ALL FAULT
W206.00 BOOL  ; ID2_READ CONDITION
W206.01 BOOL  ; START READ ID_2
W207.00 BOOL  ; POKAYOKE PLUG RELIFE FINISH
W207.01 BOOL  ; POKAYOKE PLUG RELIFE OK
W208.00 BOOL  ; CONDITION ID_@ WRITE START
W20.00 BOOL  ; SAFETY DOOR ENABLE
W20.01 BOOL  ; SHUTTER DOOR ENABLE
W20.02 BOOL  ; DUMMY DOOR ENABLE
W20.03 BOOL  ; DUMMY DOOR ENABLE END
W240.00 BOOL  ; AUTO MODE ADDITION CONDITION
W240.01 BOOL  ; AUTO MODE ADDITION CONDITION 1
W240.02 BOOL  ; AUTO CONDIRION OPEARATION P.20
W240.03 BOOL  ; AUTO ADD RUN P.20
W240.04 BOOL  ; AUTO ADD RUN P.20 CONF.
W240.05 BOOL  ; AUTO ADD RUN P.20 END
W240.06 BOOL  ; AUTO ADD RUN P.20 END CF.
W243.00 BOOL  ; ADD NEW AUTO 1 STEP REV.
W243.01 BOOL  ; ADD  AUTO CONDITION 2
W243.02 BOOL  ; AUTO CONDIRION OPEARATION P.20
W243.03 BOOL  ; AUTO CONDIRION OPEARATION P.20
W243.04 BOOL  ; AUTO ADD RUN P.20 CONF.
W243.05 BOOL  ; AUTO ADD RUN P.20 END
W243.06 BOOL  ; AUTO ADD RUN P.20 END CF.
W250.00 BOOL  ; AUTO MODE ADDITION CONDITION
W250.01 BOOL  ; AUTO MODE ADDITION CONDITION 1
W250.02 BOOL  ; AUTO CONDIRION OPEARATION P.21
W250.03 BOOL  ; AUTO ADD RUN P.21
W250.04 BOOL  ; AUTO ADD RUN P.21 CONF.
W250.05 BOOL  ; AUTO ADD RUN P.21 END
W250.06 BOOL  ; AUTO ADD RUN P.20 END CF.
W253.00 BOOL  ; AUTO MODE ADDITION CONDITION 1 REERUN
W253.01 BOOL  ; AUTO MODE ADDITION CONDITION 2 REERUN
W253.02 BOOL  ; AUTO CONDIRION OPEARATION PROGRAM REERUN
W253.03 BOOL  ; AUTO ADD RUN PROGRAM REERUN
W253.04 BOOL  ; AUTO ADD RUN PROGRAM AUTO REERUN
W253.05 BOOL  ; AUTO ADD RUN PROGRAM REERUN END
W253.06 BOOL  ; AUTO ADD RUN PROGRAM REERUN END CF
W256.00 BOOL  ; FOR INTERRUP CLEAR LAMP
W256.02 BOOL  ; PAN MARK NG CONF
W260.00 BOOL  ; FOR DIS/EN PROGRAM ADD 1STP
W260.01 BOOL  ; PB.HMI EN/DISABLE
W260.05 BOOL  ; AUTO LOOP DIS/EN P.REERUN 1STP
W260.06 BOOL  ; PB.ENNABLE/DIS 1 STEP
W260.15 BOOL  ; DISABLE MASTER CHECK
W261.00 BOOL  ; WRITE PASS WORD SET ANGLE CF.
W261.01 BOOL  ; CONF. SETUP OFFSET ANGLE
W262.00 BOOL  ; INTER RUP HOLD FAULT PICKING
W262.01 BOOL  ; CLEAR INTERRUP FAULT 375
W262.10 BOOL  ; CLEAR FAULT INTERUP
W262.11 BOOL  ; CLEAR FAULT INTER RUP 375
W273.00 BOOL  ; TRQ. WORK OK.
W273.01 BOOL  ; SENT PROGRAM N/R LEVEL 1
W273.02 BOOL  ; SENT PROGRAM N/R LEVEL 2
W273.03 BOOL  ; SENT PROGRAM N/R LEVEL 3
W273.04 BOOL  ; SENT PROGRAM N/R LEVEL 4
W273.05 BOOL  ; SENT PROGRAM N/R LEVEL 5
W273.06 BOOL  ; SENT PROGRAM N/R LEVEL 6
W273.07 BOOL  ; FOR INTERRUPT NG.AUTO NEW 1 STEP
W273.08 BOOL  ; DATA CHECK NOT LEANG STD
W273.09 BOOL  ; TRQ WORK NG
W290.00 BOOL  ; TEST
W2.00 BOOL  ; CR_EMER.STOP INTERLOCK
W2.01 BOOL  ; CR_SAFETY ENABLE
W2.02 BOOL  ; CR.DIAPHAM DOOR ENABLE
W2.03 BOOL  ; DIAPHAM DOOR ENABLE
W300.00 BOOL  ; PB_Oil Apply Down
W300.01 BOOL  ; PB Oil Apply Up
W300.02 BOOL  ; PB_Oil Apply Adv
W300.03 BOOL  ; PB_Oil Apply Ret
W30.00 BOOL  ; PB.LEARSE
W30.01 BOOL  ; PB.LEARSE
W30.02 BOOL  ; PB.RELEASE
W30.03 BOOL  ; PB.RELEASE
W310.00 BOOL  ; PL_Oil Apply Down
W310.01 BOOL  ; PL_Oil Apply Up
W310.02 BOOL  ; PL_Oil Apply Adv
W310.03 BOOL  ; PL_Oil Apply Ret
W330.00 BOOL  ; POS_Oil Apply DOWN
W330.01 BOOL  ; POS_Oil Apply UP
W330.02 BOOL  ; POS_Oil Apply ADV
W330.03 BOOL  ; POS_Oil Apply RET
W340.00 BOOL  ; PB_Oil Apply STG
W340.01 BOOL  ; PL_Oil Apply STG
W340.02 BOOL  ; PB_Oil Apply RET
W340.03 BOOL  ; PL_Oil Apply RET
W345.00 BOOL  ; Oil Apply 1 Cycle (Manual)
W345.01 BOOL  ; Oil Apply 1 Cycle (Auto)
W345.02 BOOL  ; Oil Apply 1 Cycle (Auto) Memory
W345.03 BOOL  ; Oil Apply Start Memory
W347.00 BOOL  ; M_Oil Apply Down
W347.01 BOOL  ; M_Oil Apply Up
W347.02 BOOL  ; M_Oil Apply Adv
W347.03 BOOL  ; M_Oil Apply Ret
W348.00 BOOL  ; A_Oil Apply Down
W348.01 BOOL  ; A_Oil Apply Up
W348.02 BOOL  ; A_Oil Apply Adv
W348.03 BOOL  ; A_Oil Apply Ret
W350.00 BOOL  ; OPERATION PAUSE END AUX1
W350.01 BOOL  ; OPERATION PAUSE END AUX2
W350.02 BOOL  ; OPERATION PAUSE END
W370.00 BOOL  ; PL.Auto Run Unit 1
W370.01 BOOL  ; PL.Fault Occur Unit1
W370.02 BOOL  ; PL.Auto Run Unit 2
W370.03 BOOL  ; PL.Fault Occur Unit2
W370.04 BOOL  ; PL.Auto Run Unit 3
W370.05 BOOL  ; PL.Fault Occur Unit3
W370.06 BOOL  ; PL.Auto Run Unit 4
W370.07 BOOL  ; PL.Fault Occur Unit4
W370.08 BOOL  ; PL.Auto Run Unit 5
W370.09 BOOL  ; PL.Fault Occur Unit5
W370.10 BOOL  ; PL.Auto Run Unit 6
W370.11 BOOL  ; PL.Fault Occur Unit6
W370.12 BOOL  ; PL.Auto Run Unit 7
W370.13 BOOL  ; PL.Fault Occur Unit7
W377.00 BOOL  ; PL.1st TOURQE CHECK -NG
W377.01 BOOL  ; PL.1st TOURQE CHECK OK
W377.02 BOOL  ; PL.1st TOURQE CHECK +NG
W377.03 BOOL  ; PL.1st ANGLE CHECK -NG
W377.04 BOOL  ; PL.1st ANGLE CHECK OK
W377.05 BOOL  ; PL.1st ANGLE CHECK +NG
W377.06 BOOL  ; PL.2nd TOURQE CHECK -NG
W377.07 BOOL  ; PL.2nd TOURQE CHECK OK
W377.08 BOOL  ; PL.2nd TOURQE CHECK +NG
W377.09 BOOL  ; PL.2nd ANGLE CHECK -NG
W377.10 BOOL  ; PL.2nd ANGLE CHECK OK
W377.11 BOOL  ; PL.2nd ANGLE CHECK +NG
W378.00 BOOL  ; PL.TRQ HIGH NG
W378.01 BOOL  ; PL.TRQ LOW NG
W378.02 BOOL  ; PL.ANG HIGH NG
W378.03 BOOL  ; PL.ANG LOW NG
W378.04 BOOL  ; PL.TIME MIN NG
W378.05 BOOL  ; PL.TIME MAX NG
W378.06 BOOL  ; PL.MON. TRQ HIGH NG
W378.07 BOOL  ; PL.MON. TRQ LOW NG
W378.08 BOOL  ; PL.T/R1 HIGH NG
W378.09 BOOL  ; PL.T/R1 LOW NG
W378.10 BOOL  ; PL.T/R2 HIGH NG
W378.11 BOOL  ; PL.T/R2 LOW NG
W378.12 BOOL  ; PL.BT/R HIGH NG
W378.13 BOOL  ; PL.BT/R LOW NG
W379.00 BOOL  ; CYCLE STOP ON
W3.00 BOOL  ; BZ_ALARM
W400.00 BOOL  ; MASTER CONDITION ON
W400.02 BOOL  ; MASTER ON
W400.04 BOOL  ; AUTO RUNNING
W400.05 BOOL  ; FRONT PART
W400.06 BOOL  ; FULL PART
W400.07 BOOL  ; MACHINE HOME POSITION
W401.00 BOOL  ; OPERATION-RATIO PRODUCTS COUNTING
W401.01 BOOL  ; CT1_COUNTING
W401.02 BOOL  ; CT2_COUNTING
W401.03 BOOL  ; CT3_COUNTING
W401.04 BOOL  ; CT4_COUNTING
W401.05 BOOL  ; CT5_COUNTING
W401.06 BOOL  ; CT6_COUNTING
W401.07 BOOL  ; CT7_COUNTING
W401.08 BOOL  ; CT8_COUNTING
W401.09 BOOL  ; CT9_COUNTING
W401.10 BOOL  ; CT10_COUNTING
W401.11 BOOL  ; CT11_COUNTING
W401.12 BOOL  ; CT12_COUNTING
W401.13 BOOL  ; CT13_COUNTING
W401.14 BOOL  ; CT14_COUNTING
W401.15 BOOL  ; CT15_COUNTING
W402.01 BOOL  ; T1_COUNTING
W402.02 BOOL  ; T2_COUNTING
W402.03 BOOL  ; T3_COUNTING
W402.04 BOOL  ; T4_COUNTING
W402.05 BOOL  ; T5_COUNTING
W402.06 BOOL  ; T6_COUNTING
W402.07 BOOL  ; T7_COUNTING
W405.00 BOOL  ; NORMAL ・ FAULT
W405.00 BOOL  ; MOTION FAULT CONDITION
W405.00 BOOL  ; FAULT CONDITION
W405.00 BOOL  ; FAULT CONDITION
W405.01 BOOL  ; CONDITION-OF-AUTO-START ON
W405.02 BOOL  ; CONDITION START ON 1
W405.04 BOOL  ; MANUAL CHANGE (ON BY MANUAL)
W405.05 BOOL  ; CONDITION-OF-AUTO-START ON PRESET
W406.01 BOOL  ; CT 1 UP END
W406.02 BOOL  ; CT2 COUNTING UP END
W406.03 BOOL  ; CT3 COUNTING UP END
W406.04 BOOL  ; CT4 COUNTING UP END
W406.05 BOOL  ; CT5 COUNTING UP END
W406.06 BOOL  ; CT6 COUNTING UP END
W406.07 BOOL  ; CT7 COUNTING UP END
W406.08 BOOL  ; CT8 COUNTING UP END
W407.01 BOOL  ; T1 RESET
W407.02 BOOL  ; T2 RESET
W407.03 BOOL  ; T3 RESET
W407.04 BOOL  ; T4 RESET
W407.05 BOOL  ; T5 RESET
W407.06 BOOL  ; T6 RESET
W408.01 BOOL  ; MB LOADER TIMER
W408.02 BOOL  ; MB POSITIONNING UNIT TIME OVER
W408.03 BOOL  ; DIAPHAM FEED IN UNIT TIME OVER
W408.04 BOOL  ; DIAPHAM LOADER UNIT TIME OVER
W408.05 BOOL  ; WORK TRANSFER UNIT TIME OVER
W408.06 BOOL  ; GRIPPER ROTARY UNIT TRANSFER TIME OVER
W408.07 BOOL  ; OK/NG DISCHARGE TIME OVER
W409.01 BOOL  ; CT1 RESET
W409.02 BOOL  ; CT2 RESET
W409.03 BOOL  ; CT3 RESET
W409.04 BOOL  ; CT4 RESET
W409.05 BOOL  ; CT5 RESET
W409.06 BOOL  ; CT6 RESET
W409.07 BOOL  ; CT7 RESET
W409.08 BOOL  ; CT8 RESET
W409.09 BOOL  ; CT9 RESET
W409.10 BOOL  ; CT10 RESET
W409.11 BOOL  ; CT11 RESET
W409.12 BOOL  ; CT12 RESET
W409.13 BOOL  ; CT13 RESET
W409.14 BOOL  ; CT14 RESET
W409.15 BOOL  ; CT15 RESET
W410.01 BOOL  ; CT1 COUNTING UP
W410.02 BOOL  ; CT2 COUNTING UP
W410.03 BOOL  ; CT3 COUNTING UP
W410.04 BOOL  ; CT4 COUNTING UP
W410.05 BOOL  ; CT5 COUNTING UP
W410.06 BOOL  ; CT6 COUNTING UP
W410.07 BOOL  ; CT7 COUNTING UP
W410.08 BOOL  ; CT8 COUNTING UP
W410.09 BOOL  ; CT9 COUNTING UP
W410.10 BOOL  ; CT10 COUNTING UP
W410.11 BOOL  ; CT11 COUNTING UP
W410.12 BOOL  ; CT12 COUNTING UP
W410.13 BOOL  ; CT13 COUNTING UP
W410.14 BOOL  ; CT14 COUNTING UP
W410.15 BOOL  ; CT15 COUNTING UP
W414.00 BOOL  ; MONITORING RESET
W420.09 BOOL  ; EX LOW ENERGY RUNNING COND.
W420.10 BOOL  ; EX LOW ENERGY START PERMISSION
W420.11 BOOL  ; EX FAULT CODE GROUP 1
W420.12 BOOL  ; EX FAULT CODE GROUP 2
W420.13 BOOL  ; EX FAULT CODE GROUP 3
W420.14 BOOL  ; EX COND. MODE WAIT STARTING
W420.15 BOOL  ; EX COND. MODE PAUSE
W421.00 BOOL  ; EX STOP EXTERNAL SIG. 1
W421.01 BOOL  ; EX STOP EXTERNAL SIG. 2
W421.02 BOOL  ; EX STOP EXTERNAL SIG. 3
W421.03 BOOL  ; EX STOP EXTERNAL SIG. 4
W421.04 BOOL  ; EX STOP EXTERNAL SIG. 5
W421.05 BOOL  ; EX START･BREAK EXTERNAL SIG. 1
W421.06 BOOL  ; EX START･BREAK EXTERNAL SIG. 2
W421.07 BOOL  ; EX START･BREAK EXTERNAL SIG. 3
W421.08 BOOL  ; EX START･BREAK EXTERNAL SIG. 4
W421.09 BOOL  ; EX START･BREAK EXTERNAL SIG. 5
W422.11 BOOL  ; EX LOW ENERGY START CONFIRM.
W422.12 BOOL  ; CR LOW ENERGY OUTPUT 1
W422.13 BOOL  ; CR LOW ENERGY OUTPUT 2
W422.14 BOOL  ; CR LOW ENERGY OUTPUT 3
W422.15 BOOL  ; CR LOW ENERGY OUTPUT 4
W423.00 BOOL  ; CR LOW ENERGY OUTPUT 5
W423.04 BOOL  ; EX ENERGY SAVING
W424.00 BOOL  ; OUTPUT 1 START CONFIRM.
W424.01 BOOL  ; OUTPUT 1 <SETTING> 0 IN DELAY TIME OF BEGINNING
W424.02 BOOL  ; OUTPUT 1 START DELAY COMPL.
W424.03 BOOL  ; OUTPUT 1 <SETTING> 0 IN LOW ENERGY TIME
W424.04 BOOL  ; OUTPUT 1 LOW ENERGY END
W424.05 BOOL  ; OUTPUT 1 LOW ENERGY START AUXILIARY
W424.06 BOOL  ; OUTPUT 1 EXTERNAL START AUXILIARY
W424.07 BOOL  ; OUTPUT 1 BREAK START
W424.08 BOOL  ; OUTPUT 1 <SETTING> 0 IN INTERRUPTION DELAY TIME
W424.09 BOOL  ; OUTPUT 1 START BREAK END
W424.10 BOOL  ; OUTPUT 1 FAULT STOP START
W424.14 BOOL  ; OUTPUT 1 EXTERNAL BEGINNING, 1 SHOT, AND AUX.
W424.15 BOOL  ; OUTPUT 1 INTERRUPTION BEGINNING, 1 SHOT, AND AUX.
W425.00 BOOL  ; OUTPUT 2 START CONFIRM.
W425.01 BOOL  ; OUTPUT 2 <SETTING> 0 IN DELAY TIME OF BEGINNING
W425.02 BOOL  ; OUTPUT 2 START DELAY COMPL.
W425.03 BOOL  ; OUTPUT 2 <SETTING> 0 IN LOW ENERGY TIME
W425.04 BOOL  ; OUTPUT 2 LOW ENERGY END
W425.05 BOOL  ; OUTPUT 2 LOW ENERGY START AUXILIARY
W425.06 BOOL  ; OUTPUT 2 EXTERNAL START AUXILIARY
W425.07 BOOL  ; OUTPUT 2 BREAK START
W425.08 BOOL  ; OUTPUT 2 <SETTING> 0 IN INTERRUPTION DELAY TIME
W425.09 BOOL  ; OUTPUT 2 START BREAK END
W425.10 BOOL  ; OUTPUT 2 FAULT STOP START
W425.14 BOOL  ; OUTPUT 2 EXTERNAL BEGINNING, 1 SHOT, AND AUX.
W425.15 BOOL  ; OUTPUT 2 INTERRUPTION BEGINNING, 1 SHOT, AND AUX.
W426.00 BOOL  ; OUTPUT 3 START CONFIRM.
W426.01 BOOL  ; OUTPUT 3 <SETTING> 0 IN DELAY TIME OF BEGINNING
W426.02 BOOL  ; OUTPUT 3 START DELAY COMPL.
W426.03 BOOL  ; OUTPUT 3 <SETTING> 0 IN LOW ENERGY TIME
W426.04 BOOL  ; OUTPUT 3 LOW ENERGY END
W426.05 BOOL  ; OUTPUT 3 LOW ENERGY START AUXILIARY
W426.06 BOOL  ; OUTPUT 3 EXTERNAL START AUXILIARY
W426.07 BOOL  ; OUTPUT 3 BREAK START
W426.08 BOOL  ; OUTPUT 3 <SETTING> 0 IN INTERRUPTION DELAY TIME
W426.09 BOOL  ; OUTPUT 3 START BREAK END
W426.10 BOOL  ; OUTPUT 3 FAULT STOP START
W426.14 BOOL  ; OUTPUT 3 EXTERNAL BEGINNING, 1 SHOT, AND AUX.
W426.15 BOOL  ; OUTPUT 3 INTERRUPTION BEGINNING, 1 SHOT, AND AUX.
W427.00 BOOL  ; OUTPUT 4 START CONFIRM.
W427.01 BOOL  ; OUTPUT 4 <SETTING> 0 IN DELAY TIME OF BEGINNING
W427.02 BOOL  ; OUTPUT 4 START DELAY COMPL.
W427.03 BOOL  ; OUTPUT 4 <SETTING> 0 IN LOW ENERGY TIME
W427.04 BOOL  ; OUTPUT 4 LOW ENERGY END
W427.05 BOOL  ; OUTPUT 4 LOW ENERGY START AUXILIARY
W427.06 BOOL  ; OUTPUT 4 EXTERNAL START AUXILIARY
W427.07 BOOL  ; OUTPUT 4 BREAK START
W427.08 BOOL  ; OUTPUT 4 <SETTING> 0 IN INTERRUPTION DELAY TIME
W427.09 BOOL  ; OUTPUT 4 START BREAK END
W427.10 BOOL  ; OUTPUT 4 FAULT STOP START
W427.14 BOOL  ; OUTPUT 4 EXTERNAL BEGINNING, 1 SHOT, AND AUX.
W427.15 BOOL  ; OUTPUT 4 INTERRUPTION BEGINNING, 1 SHOT, AND AUX.
W428.00 BOOL  ; OUTPUT 5 START CONFIRM.
W428.01 BOOL  ; OUTPUT 5 <SETTING> 0 IN DELAY TIME OF BEGINNING
W428.02 BOOL  ; OUTPUT 5 START DELAY COMPL.
W428.03 BOOL  ; OUTPUT 5 <SETTING> 0 IN LOW ENERGY TIME
W428.04 BOOL  ; OUTPUT 5 LOW ENERGY END
W428.05 BOOL  ; OUTPUT 5 LOW ENERGY START AUXILIARY
W428.06 BOOL  ; OUTPUT 5 EXTERNAL START AUXILIARY
W428.07 BOOL  ; OUTPUT 5 BREAK START
W428.08 BOOL  ; OUTPUT 5 <SETTING> 0 IN INTERRUPTION DELAY TIME
W428.09 BOOL  ; OUTPUT 5 START BREAK END
W428.10 BOOL  ; OUTPUT 5 FAULT STOP START
W428.14 BOOL  ; OUTPUT 5 EXTERNAL BEGINNING, 1 SHOT, AND AUX.
W428.15 BOOL  ; OUTPUT 5 INTERRUPTION BEGINNING, 1 SHOT, AND AUX.
W430.00 BOOL  ; LOW ENERGY AUTO
W430.01 BOOL  ; CUMULATE TIME RESET
W430.02 BOOL  ; LOW ENERGY AUTOMATIC CHANGE
W430.03 BOOL  ; LOW ENERGY AUTOMATIC CHANGE
W431.00 BOOL  ; MANUAL START PB
W431.01 BOOL  ; MANUAL LOW ENERGY START
W431.02 BOOL  ; ON SWITCHING RESET
W431.03 BOOL  ; OFF SWITCHING RESET
W433.00 BOOL  ; PB OUTPUT 1 START
W433.01 BOOL  ; PB OUTPUT 2 START
W433.02 BOOL  ; PB OUTPUT 3 START
W433.03 BOOL  ; PB OUTPUT 4 START
W433.04 BOOL  ; PB OUTPUT 5 START
W435.00 BOOL  ; OUTPUT 1 START DELAY TIME
W435.01 BOOL  ; OUTPUT 1 LOW ENERGY TIME
W435.02 BOOL  ; OUTPUT 1 BREAK DELAY TIME
W435.03 BOOL  ; OUTPUT 1 RESET
W435.04 BOOL  ; OUTPUT 1 ACCUMULATION CT_m RESET
W436.00 BOOL  ; OUTPUT 2 START DELAY TIME
W436.01 BOOL  ; OUTPUT 2 LOW ENERGY TIME
W436.02 BOOL  ; OUTPUT 2 BREAK DELAY TIME
W436.03 BOOL  ; OUTPUT 2 RESET
W436.04 BOOL  ; OUTPUT 2 ACCUMULATION CT_m RESET
W437.00 BOOL  ; OUTPUT 3 START DELAY TIME
W437.01 BOOL  ; OUTPUT 3 LOW ENERGY TIME
W437.02 BOOL  ; OUTPUT 3 BREAK DELAY TIME
W437.03 BOOL  ; OUTPUT 3 RESET
W437.04 BOOL  ; OUTPUT 3 ACCUMULATION CT_m RESET
W438.00 BOOL  ; OUTPUT 4 START DELAY TIME
W438.01 BOOL  ; OUTPUT 4 LOW ENERGY TIME
W438.02 BOOL  ; OUTPUT 4 BREAK DELAY TIME
W438.03 BOOL  ; OUTPUT 4 RESET
W438.04 BOOL  ; OUTPUT 4 ACCUMULATION CT_m RESET
W439.00 BOOL  ; OUTPUT 5 START DELAY TIME
W439.01 BOOL  ; OUTPUT 5 LOW ENERGY TIME
W439.02 BOOL  ; OUTPUT 5 BREAK DELAY TIME
W439.03 BOOL  ; OUTPUT 5 RESET
W439.04 BOOL  ; OUTPUT 5 ACCUMULATION CT_m RESET
W440.00 BOOL  ; MODEL SELECTED END
W450.08 BOOL  ; PB_FAULT RESET
W450.09 BOOL  ; PB_BZ.RESET
W456.00 BOOL  ; PL.DISCHARGE PROCESS
W456.01 BOOL  ; PB Discharge
W456.02 BOOL  ; PB.DISCHARGE
W456.03 BOOL  ; PB.MODEL SELECTED
W457.02 BOOL  ; PL.DISCHARGE
W457.03 BOOL  ; PL.DISCHARGE
W461.00 BOOL  ; PB.MD LOAD IN DOWN
W461.01 BOOL  ; PB.MD LOAD IN UP
W461.02 BOOL  ; PB.MD LOAD OUT DOWN
W461.03 BOOL  ; PB.MD LOAD OUT UP
W461.04 BOOL  ; PB.MB LOAD OUT UNIT DOWN
W461.05 BOOL  ; PB.MB LOAD OUT UNIT UP
W461.06 BOOL  ; PB.MAG HOLDER 1 MAGNET
W461.07 BOOL  ; PB.MAG HOLDER 1 DE-MAGNET
W461.08 BOOL  ; PB.MAG HOLDER 2 MAGNET
W461.09 BOOL  ; PB.MAG HOLDER 2 DE-MAGNET
W461.10 BOOL  ; PB.MB LOAD UNIT ADV
W461.11 BOOL  ; PB.MB LOAD UNIT RET
W461.12 BOOL  ; PB.WORK ROTATE START
W461.13 BOOL  ; PB.WORK ROTATE SLOW
W461.14 BOOL  ; PB.PIN UP
W461.15 BOOL  ; PB.PIN DOWN
W462.00 BOOL  ; PB.laod bwd
W462.01 BOOL  ; PB.Load FWD (home)
W462.02 BOOL  ; PB.JIG CHANGE OVER MIRROR
W462.03 BOOL  ; PB.JIG CHANGE OVER NORMAL
W462.04 BOOL  ; PB.N/R CHANGE OVER MIRROR
W462.05 BOOL  ; PB.N/R CHANGE OVER NORMAL
W462.06 BOOL  ; PB.WORK CLAMP CHANGE OVER MIRROR
W462.07 BOOL  ; PB.WORK CLAMP CHANGE OVER NORMAL
W462.12 BOOL  ; PB.OIL SUPPLY ON
W462.13 BOOL  ; PB.OIL SUPPLY OFF
W462.14 BOOL  ; ID WRITE
W462.15 BOOL  ; ID READ
W463.01 BOOL  ; PB. SAFETY COVER OUT DOWN
W463.02 BOOL  ; PB.SAFETY COVER IN UP
W463.03 BOOL  ; PB.SAFETY COVER IN DOWN
W463.04 BOOL  ; PB.1EC3 ADV.
W463.05 BOOL  ; PB.1EC3 RET.
W463.06 BOOL  ; PB.GRIPPER 1 CHUCK
W463.07 BOOL  ; PB.GRIPPER 1 UNCHUCK
W463.08 BOOL  ; PB.GRIPPER 2 CHUCK
W463.09 BOOL  ; PB.GRIPPER 2 UNCHUCK
W463.10 BOOL  ; PB.GRIPPER 3 CHUCK
W463.11 BOOL  ; PB.GRIPPER 3 UNCHUCK
W463.12 BOOL  ; PB.GRIPPER UNIT DOWN
W463.13 BOOL  ; PB.GRIPPER UNIT UP
W463.14 BOOL  ; PB.1EC3 MID.
W464.00 BOOL  ; PB.FLIP 180
W464.01 BOOL  ; PB.FLIP 0
W464.02 BOOL  ; PB.1EC4 LOADER UNIT ADV
W464.03 BOOL  ; PB.1EC4 LOADER UNIT RET
W465.00 BOOL  ; PB.SLIDE TRANSFER ADV.
W465.01 BOOL  ; PB.SLIDE TRANSFER RET.
W465.02 BOOL  ; PB. PUSHER DOWN
W465.03 BOOL  ; PB. PUSHER UP
W465.07 BOOL  ; PB. MASTER CHECK START
W465.09 BOOL  ; PB. MASTER CHECK START
W465.12 BOOL  ; PB GD-P2S SEL.
W465.13 BOOL  ; PB. GD-P3SH SEL
W467.00 BOOL  ; PB.1EC1 DOWN
W467.01 BOOL  ; PB.1EC1 UP
W467.02 BOOL  ; PB.GRIPPER 1 CHUCK
W467.03 BOOL  ; PB.GRIPPER 1 UNCHUCK
W467.04 BOOL  ; PB.GRIPPPER 2 CHUCK
W467.05 BOOL  ; PB.GRIPPPER 2 UNCHUCK
W467.06 BOOL  ; PB.ROTATE GRIP UNIT 180
W467.07 BOOL  ; PB.ROTATE GRIP UNIT 0
W467.08 BOOL  ; PB.GRIPPER 1 UNIT ADV
W467.09 BOOL  ; PB.GRIPPER 1 UNIT RET
W467.10 BOOL  ; PB.GRIPPER 2 UNIT ADV
W467.11 BOOL  ; PB.GRIPPER 2 UNIT RET
W468.06 BOOL  ; FLoat sensor
W469.00 BOOL  ; PB.DISCH PALLET DOWN
W469.01 BOOL  ; PB.DISCH PALLET UP
W469.02 BOOL  ; PB.OK PUSH UP
W469.03 BOOL  ; PB.OK PULL DOWN
W469.04 BOOL  ; PB.NG PULL DOWN
W469.05 BOOL  ; PB.NG PUSH UP
W470.09 BOOL  ; WORK SLIDE TRANSFER HOME
W475.00 BOOL  ; PB.DATA READ
W475.01 BOOL  ; PB.DATA REGIS.
W477.00 BOOL  ; PB.MEMORY REAET
W477.01 BOOL  ; PB.SKIP ID ON
W477.02 BOOL  ; PB.SKIP ID OFF
W477.04 BOOL  ; PB.1EC1 BREAK RELEASE
W477.05 BOOL  ; PB.1EC2 BREAK RELEASE
W477.06 BOOL  ; PB.1EC3 BREAK RELEASE
W477.07 BOOL  ; PB.1EC4 BREAK RELEASE
W477.08 BOOL  ; DISABLE MASTER CHECK
W477.11 BOOL  ; PB.STOPPER CONVEYOR NO USE
W478.00 BOOL  ; P11-12 1 Cycle Start
W478.01 BOOL  ; P13-14 1 Cycle Start
W478.02 BOOL  ; P15 1 Cycle Start
W478.03 BOOL  ; P16 1 Cycle Start
W478.04 BOOL  ; P17 1 Cycle Start
W478.07 BOOL  ; PB. MB LOADER UNIT /ROTATE HOME
W478.07 BOOL  ; UNIT1 HOME POS.
W478.08 BOOL  ; PB.DIAPH HOME
W478.09 BOOL  ; PB.TRANSFER RETURN
W478.10 BOOL  ; PB.ROTARY GRIP UNIT HOME
W478.11 BOOL  ; PB.DISCHARGE HOME
W478.15 BOOL  ; PB all unit home
W479.01 BOOL  ; P14 1 cycle run
W479.06 BOOL  ; DIAPH FEED UNIT HOME POS.(DISCHARGE)
W479.07 BOOL  ; MB LOAD UNIT HOME POS.
W479.08 BOOL  ; HORN ROTATE UNIT HOME POS. 1 (NG POS.)
W479.09 BOOL  ; wORK SLIDE TRANSFER
W479.10 BOOL  ; WORK Rotary Transfer Home
W479.11 BOOL  ; OK/NG DISCH HOME
W479.12 BOOL  ; ROTARY GRIPPER UNIT HOME POS.1
W479.13 BOOL  ; OIL APPLY UNIT HOME POS.
W479.14 BOOL  ; MB WORK UNIT HOME POS. (OK POS.)
W479.15 BOOL  ; ROTARY GRIPPER UNIT HOME POS.2
W480.07 BOOL  ; PL UNIT 1 HOME
W480.08 BOOL  ; Diaph unit Home
W481.00 BOOL  ; MASTER CONDITION 1:PC GOOD
W481.01 BOOL  ; MASTER CONDITION 2:PRESSURE NORMAL
W481.02 BOOL  ; MASTER CONDITION 3:FUSE NORMAL
W481.03 BOOL  ; MASTER CONDITION 4:SAFETY SLIDE CLOSE
W481.04 BOOL  ; MASTER CONDITION 5:SAFETY COVER CLOSE
W481.05 BOOL  ; MASTER CONDITION 6
W481.06 BOOL  ; MASTER CONDITION 7
W481.07 BOOL  ; MASTER CONDITION 8
W481.08 BOOL  ; MASTER CONDITION 9:EMG STOP NO PRSS
W481.09 BOOL  ; MASTER CONDITION 10:NO EMG FAULT
W481.10 BOOL  ; USE IS IMPOSSIBLE.   1
W481.11 BOOL  ; USE IS IMPOSSIBLE.   2
W481.12 BOOL  ; USE IS IMPOSSIBLE.   3
W481.13 BOOL  ; USE IS IMPOSSIBLE.   4
W481.14 BOOL  ; USE IS IMPOSSIBLE.   5
W481.15 BOOL  ; USE IS IMPOSSIBLE.   6
W482.00 BOOL  ; START CONDITION 1-1:HOME POS.
W482.01 BOOL  ; START CONDITION 1-2: AUTO MODE
W482.02 BOOL  ; START CONDITION 1-3:WORK NOT FULL
W482.02 BOOL  ; START CONDITION 1-3
W482.03 BOOL  ; START CONDITION 1-4:NG BOX NOT FULL
W482.04 BOOL  ; START CONDITION 1-5:EC NORMAL
W482.05 BOOL  ; START CONDITION 1-6:DOOR NOT ENABLE
W482.06 BOOL  ; START CONDITION 1-7:MTD1 NORMAL
W482.07 BOOL  ; START CONDITION 1-8
W482.08 BOOL  ; START CONDITION 1-9
W482.09 BOOL  ; START CONDITION 1-10
W482.10 BOOL  ; START CONDITION 1-11
W482.11 BOOL  ; START CONDITION 1-12
W482.12 BOOL  ; START CONDITION 1-13:NO FAULT ALL
W482.13 BOOL  ; START CONDITION 1-14
W482.14 BOOL  ; USE IS IMPOSSIBLE.   1-1
W482.15 BOOL  ; USE IS IMPOSSIBLE.   1-2
W483.00 BOOL  ; START CONDITION 2-1:FCK EMER OK
W483.01 BOOL  ; START CONDITION 2-2: FCK  FUSE OK
W483.02 BOOL  ; START CONDITION 2-3: FCK MASTER ON
W483.03 BOOL  ; START CONDITION 2-4: FINAL ALL HOME
W483.04 BOOL  ; START CONDITION 2-5: FCK AUTO RUN
W483.05 BOOL  ; START CONDITION 2-6
W483.06 BOOL  ; START CONDITION 2-7
W483.07 BOOL  ; START CONDITION 2-8
W483.08 BOOL  ; START CONDITION 2-9
W483.09 BOOL  ; START CONDITION 2-10
W483.10 BOOL  ; START CONDITION 2-11
W483.11 BOOL  ; START CONDITION 2-12
W483.12 BOOL  ; START CONDITION 2-13
W483.13 BOOL  ; START CONDITION 2-14:FCK NO FAULT
W483.14 BOOL  ; USE IS IMPOSSIBLE.   2-1
W483.15 BOOL  ; USE IS IMPOSSIBLE.   2-2
W484.00 BOOL  ; PL.MB LOAD IN DOWN
W484.01 BOOL  ; PL.MB LOAD IN UP
W484.02 BOOL  ; PL.MB LOAD OUT DOWN
W484.03 BOOL  ; PL.MB LOAD OUT UP
W484.04 BOOL  ; PL.MB LOAD OUT UNIT DOWN
W484.05 BOOL  ; PL.MB LOAD OUT UNIT UP
W484.06 BOOL  ; PL.MB MG1 MAGNETIZE
W484.07 BOOL  ; PL.MB MG1 DE-MAGNETIZE
W484.08 BOOL  ; PL.MB MG2 MAGNETIZE
W484.09 BOOL  ; PL.MB MG2 DE-MAGNETIZE
W484.10 BOOL  ; PL.MB LOAD UNIT ADV
W484.11 BOOL  ; PL.MB LOAD UNIT RET
W484.12 BOOL  ; PL.MB ROTATE
W484.13 BOOL  ; PL.PL.MB ROTATE STOP
W484.14 BOOL  ; PL.PIN UP
W484.15 BOOL  ; PL.PIN DOWN
W485.00 BOOL  ; PL.TIGHT SLIDE2 RET.[102]
W485.01 BOOL  ; PL.TIGHT SLIDE2 ADV.[103]
W485.02 BOOL  ; PL.JIG CHANGE OVER MIRROR[114]
W485.03 BOOL  ; PL.JIG CHANGE OVER NORMAL[115]
W485.04 BOOL  ; PL.N/R CHANGE OVER MIRROR[200]
W485.05 BOOL  ; PL.N/R CHANGE OVER NORMAL[201]
W485.06 BOOL  ; PL.WORK CLAMP CHANGE OVER MIRROR[202]
W485.07 BOOL  ; PL.WORK CLAMP CHANGE OVER NORMAL[203]
W485.12 BOOL  ; PL.OIL SUPPLY MOTOR ON[]
W485.13 BOOL  ; PL.OIL SUPPLY MOTOR OFF[]
W485.14 BOOL  ; IND CHECK NG
W485.15 BOOL  ; IND CHECK OK
W486.00 BOOL  ; PL. SAFETY COVER OUT UP
W486.01 BOOL  ; PL. SAFETY COVER OUT DOWN
W486.02 BOOL  ; PL. SAFETY COVER IN UP
W486.03 BOOL  ; PL. SAFETY COVER IN DOWN
W486.04 BOOL  ; PL.1EC3 DIAPHAM LOADER ADV
W486.05 BOOL  ; PL.1EC3 DIAPHAM LOADER RET
W486.06 BOOL  ; PL.GRIPPER 1 CHUCK
W486.07 BOOL  ; PL.GRIPPER 1 UNCHUCK
W486.08 BOOL  ; PL.GRIPPER 2 CHUCK
W486.09 BOOL  ; PL.GRIPPER 2 UNCHUCK
W486.10 BOOL  ; PL.GRIPPER 3 CHUCK
W486.11 BOOL  ; PL.GRIPPER 3 UNCHUCK
W486.12 BOOL  ; PL.GRIPPER UNIT DOWN
W486.13 BOOL  ; PL.GRIPPER UNIT UP
W486.14 BOOL  ; PL.1EC3 DIAPHAM LOADER MID
W487.00 BOOL  ; PL.180 FLIP ADV
W487.01 BOOL  ; PL.180 FLIP RET
W487.02 BOOL  ; PL.1EC4 LOAD UNIT ADV.
W487.03 BOOL  ; PL.1EC4 LOAD UNIT RET.
W488.00 BOOL  ; PL.TRANSFER SLIDE ADV.
W488.01 BOOL  ; PL.TRANSFER SLIDE RET
W488.02 BOOL  ; PL. WORK PUSHER DOWN
W488.03 BOOL  ; PL. WORK PUSHER UP
W488.09 BOOL  ; PL. MASTER CHECK START
W488.12 BOOL  ; PL. GD-P3S SEL
W488.13 BOOL  ; PL. GD-P3SH SEL
W488.14 BOOL  ; IND CHECK NG
W488.15 BOOL  ; IND CHECK OK
W490.00 BOOL  ; PL.1EC1 ROTARY GRIP DOWN
W490.01 BOOL  ; PL.1EC1 ROTARY GRIP UP
W490.02 BOOL  ; PL.GRIPPER 1 CHUCK
W490.03 BOOL  ; PL.GRIPPER 1 UNCHUCK
W490.04 BOOL  ; PL.GRIPPER 2 CHUCK
W490.05 BOOL  ; PL.GRIPPER 2 UNCHUCK
W490.06 BOOL  ; PL.FLIP 180
W490.07 BOOL  ; PL.FLIP 0
W490.08 BOOL  ; PL.GRIPPER 1 UNIT ADV
W490.09 BOOL  ; PL.GRIPPER 1 UNIT RET
W490.10 BOOL  ; PL.GRIPPER 2 UNIT ADV
W490.11 BOOL  ; PL.GRIPPER 2 UNIT RET
W491.01 BOOL  ; mem master ok
W492.00 BOOL  ; PL.DISCHARGE PALLET DOWN
W492.01 BOOL  ; PL.DISCHARGE PALLET UP
W492.02 BOOL  ; PL.OK PUSH
W492.03 BOOL  ; PL.OK PULL
W492.04 BOOL  ; PL.NG PULL
W492.05 BOOL  ; PL.NG PUSH
W498.00 BOOL  ; PL.DATA READ
W498.01 BOOL  ; PL.DATA REGIS.
W499.01 BOOL  ; pb ct history clear
W499.02 BOOL  ; NG.CT 2 RESET
W499.03 BOOL  ; NG.CT 3 RESET
W499.04 BOOL  ; NG.CT 4 RESET
W4.01 BOOL  ; MASTER OFF CONF. AUX.
W500.00 BOOL  ; PL MEMORY RESET DONE
W500.01 BOOL  ; PL. ID SKIP ON
W500.04 BOOL  ; PL.EC1 RELEASE CONF
W500.05 BOOL  ; PL.EC2 RELEASE CONF
W500.06 BOOL  ; PL.EC3 RELEASE CONF
W500.07 BOOL  ; PL.EC4 RELEASE CONF
W500.08 BOOL  ; LAMP OFF OLD // LAMP ON NEW ID2 MAP
W500.09 BOOL  ; LAMP OFF OLD // LAMP ON NEW ID MAP
W500.11 BOOL  ; PL.STOPPER CONVEYOR NO USE
W501.00 BOOL  ; MF001_SHUTTER 1 OPERATION FAULT
W501.01 BOOL  ; MF002_SHUTTER 2 OPERATION FAULT
W501.02 BOOL  ; MF003_DIAPH GRIPPER UNIT OPERATION FAULT
W501.03 BOOL  ; MF004_DIAPH GRIPPER 1 OPERATION FAULT
W501.04 BOOL  ; MF005_DIAPH GRIPPER 2 OPERATION FAULT
W501.05 BOOL  ; MF006_DIAPH GRIPPER 3 OPERATION FAULT
W501.06 BOOL  ; MF007_DIAPH GRIPPER FLIP OPERATION FAULT
W501.07 BOOL  ; MF008_ROTARY GRIPPER 1 OPERATION FAULT
W501.08 BOOL  ; MF009_ROTARY GRIPPER 2 OPERATION FAULT
W501.09 BOOL  ; MF010_ROTARY GRIPPER UNIT 1 OPERATION FAULT
W501.10 BOOL  ; MF011_ROTARY GRIPPER UNIT 2 OPERATION FAULT
W501.11 BOOL  ; MF012_MB LOAD IN OPERATION FAULT
W501.12 BOOL  ; MF013_MB LOAD OUT OPERATION FAULT
W501.13 BOOL  ; MF014_MB LOAD OUT UNIT OPERATION FAULT
W501.14 BOOL  ; MF015_MB SLIDE UNIT OPERATION FAULT
W501.15 BOOL  ; MF016_MB POSITION PIN UNIT OPERATION FAULT
W502.00 BOOL  ; MF017_WORK TRANSFER UNIT OPERATION FAULT
W502.01 BOOL  ; MF018_FINISH TRAY OPERATION FAULT
W502.02 BOOL  ; MF019_OK PUSH OPERATION FAULT
W502.03 BOOL  ; MF020_NG PULL OPERATION FAULT
W502.04 BOOL  ; -
W502.05 BOOL  ; -
W505.00 BOOL  ; FAULT 365 SKIP PROCESS O/P
W505.01 BOOL  ; FAULT 366 ID2 TACK NG
W505.02 BOOL  ; FAULT 367 SUMCHECK ERROR
W505.03 BOOL  ; FAULT_368 ID-TAC ERROR
W505.04 BOOL  ; FAULT369_PLUG ASSY ID2 NOT COMPLETE
W505.05 BOOL  ; FAULT_370 ID-TAC READ ERROR
W505.06 BOOL  ; FAULT_371 REPEAT PROCESS ID2
W505.07 BOOL  ; FAULT_372 SOL.OIL FAULT
W505.08 BOOL  ; FAULT_373 SKIP PROCESS PICKKING
W505.09 BOOL  ; FAULT 374 SENSOR CLEAR FAULT ABNORMAL
W505.10 BOOL  ; FAULT 375 PICKKING SENSER DOUBLE PROCESS
W505.11 BOOL  ; FAULT 376 PLUG MODEL MISSTAKE
W505.12 BOOL  ; FAULT377 NG TRAY FULL
W505.13 BOOL  ; FAULT 378 GD-P3S MASTER WRONG TYPE
W505.14 BOOL  ; FAULT 379 GD-P3SH MASTER WRONG TYPE
W505.15 BOOL  ; FAULT 380 MASTER NG
W506.00 BOOL  ; FAULT 381MASTER DOES NOT TAKEN
W506.01 BOOL  ; FAULT 382 MASTER MISTAKE
W50.00 BOOL  ; ALL UNIT HOME POS.
W510.00 BOOL  ; UNLATCH
W510.01 BOOL  ; UNIT1 UNLATCH
W510.02 BOOL  ; UNIT2 UNLATCH
W510.03 BOOL  ; UNIT3 UNLATCH
W510.04 BOOL  ; UNIT4 UNLATCH
W510.05 BOOL  ; UNIT5 UNLATCH
W510.06 BOOL  ; UNIT6 UNLATCH
W510.07 BOOL  ; UNIT7 UNLATCH
W511.00 BOOL  ; MASTER(AIR) ON BUTTON
W511.01 BOOL  ; AUTOMATIC-START BUTTON
W511.02 BOOL  ; CYCLE-STOP BUTTON
W511.03 BOOL  ; DATA INDICATION
W511.04 BOOL  ; FEW ENERGY RUNNING
W511.05 BOOL  ; FEW ENERGY AUTOMATIC
W511.06 BOOL  ; NG  TWICE CONTINOUS
W511.07 BOOL  ; FAULT 200 CONDITION
W511.08 BOOL  ; MOTION FAULT CONDITION
W511.09 BOOL  ; RESET
W511.10 BOOL  ; CYCLE TIME MEASUREMENT TIMING
W511.11 BOOL  ; WATCH_DOG_OK
W511.12 BOOL  ; EQUIPMENT STOPPING
W511.13 BOOL  ; PC GOOD
W55.00 BOOL  ; IND.MB LOAD IN DOWN
W55.01 BOOL  ; PB.MB LOAD IN UP
W55.02 BOOL  ; IND.MB LOAD OUT DOWN
W55.03 BOOL  ; IND.MB LOAD OUT UP
W55.04 BOOL  ; IND.MB LOAD OUT UNIT DOWN
W55.05 BOOL  ; IND.MB LOAD OUT UNIT UP
W55.06 BOOL  ; IND.MAG HOLDER 1 MAGNET
W55.07 BOOL  ; IND.MAG HOLDER 1 DE-MAGNET
W55.08 BOOL  ; IND.MAG HOLDER 2 MAGNET
W55.09 BOOL  ; IND.MAG HOLDER 2 DE-MAGNET
W55.10 BOOL  ; IND.MB LOAD UNIT ADV
W55.11 BOOL  ; IND.MB LOAD UNIT RET
W55.12 BOOL  ; IND.WORK ROTATE START
W55.13 BOOL  ; IND.WORK ROTATE INPOSITION
W55.14 BOOL  ; IND.PIN UP
W55.15 BOOL  ; PB.PIN DOWN
W56.01 BOOL  ; IND.SAFETY COVER 1 DOWN
W56.02 BOOL  ; IND.SAFETY COVER 2 UP
W56.03 BOOL  ; IND.SAFETY COVER 2 DOWN
W56.04 BOOL  ; IND.1EC3 ADV.
W56.05 BOOL  ; IND.1EC3 RET.
W56.06 BOOL  ; IND.GRIPPER 1 CHUCK
W56.07 BOOL  ; IND.GRIPPER 1 UNCHUCK
W56.08 BOOL  ; IMD.GRIPPER 2 CHUCK
W56.09 BOOL  ; IND.GRIPPER 2 UNCHUCK
W56.10 BOOL  ; IND.GRIPPER 3 CHUCK
W56.11 BOOL  ; IND.GRIPPER 3 UNCHUCK
W56.12 BOOL  ; IND.GRIPPER UNIT DOWN
W56.13 BOOL  ; IND.GRIPPER UNIT UP
W56.14 BOOL  ; IND.1EC3 MID.
W57.00 BOOL  ; IND.FLIP 180
W57.01 BOOL  ; IND.FLIP 0
W57.02 BOOL  ; IND.1EC4 LOADER UNIT ADV
W57.03 BOOL  ; INd.1EC4 LOADER UNIT RET
W57.04 BOOL  ; STOPPER 1 DOWN
W57.05 BOOL  ; STOPPEER 1 UP
W57.06 BOOL  ; STOPPER 2 DOWN
W57.07 BOOL  ; STOPPER 2 UP
W57.08 BOOL  ; STOPPER 3 DOWN
W57.09 BOOL  ; STOPPER 3 UP
W57.10 BOOL  ; WORK PUSHER UP
W57.11 BOOL  ; WORK PUSHER DOWN
W57.12 BOOL  ; NAGARA SWITCH
W58.00 BOOL  ; IND.SLIDE TRANSFER ADV.
W58.01 BOOL  ; IND.SLIDE TRANSFER RET.
W5.01 BOOL  ; FAULT EMG.STOP
W5.02 BOOL  ; FAULT AUTO STOP
W5.03 BOOL  ; FAULT CYCLE STOP
W5.04 BOOL  ; FAULT STOP ALL
W5.05 BOOL  ; OTHER FAULT
W60.00 BOOL  ; IND.1EC1 DOWN
W60.01 BOOL  ; IND.1EC1 UP
W60.02 BOOL  ; IND.GRIPPER 1 CHUCK
W60.03 BOOL  ; IND.GRIPPER 1 UNCHUCK
W60.04 BOOL  ; IND.GRIPPPER 2 CHUCK
W60.05 BOOL  ; IND.GRIPPER 2 UNCHUCK
W60.06 BOOL  ; IND.ROTATE GRIP UNIT 180
W60.07 BOOL  ; IND.ROTATE GRIP UNIT 0
W60.08 BOOL  ; IND.GRIPPER 1 UNIT ADV
W60.09 BOOL  ; IND.GRIPPER 1 UNIT RET
W60.10 BOOL  ; IND.GRIPPER 2 UNIT ADV
W60.11 BOOL  ; IND.GRIPPER 2 UNIT RET
W61.00 BOOL  ; IND.DISCH PALLET DOWN
W61.01 BOOL  ; IND.DISCH PALLET UP
W61.02 BOOL  ; IND.OK PUSH UP
W61.03 BOOL  ; IND.OK PULL DOWN
W61.04 BOOL  ; IND.NG PULL DOWN
W61.05 BOOL  ; PB.NG PUSH UP
W65.00 BOOL  ; IND.SAFETY COVER OPEN
W65.01 BOOL  ; IND.DUMMY FRANGE1,2 CLAMP
W65.02 BOOL  ; IND.DUMMY FRANGE1,2 UN-CLAMP
W65.03 BOOL  ; IND.TIGHTENING SLIDE1 TIGHT
W65.04 BOOL  ; IND.TIGHTENING SLIDE1 HOME
W65.05 BOOL  ; IND.TIGHTENING SLIDE2 ADV.
W65.06 BOOL  ; IND.TIGHTENING SLIDE2 RET.
W65.07 BOOL  ; IND.WORK CLAMP1,2 DOWN
W65.08 BOOL  ; IND.WORK CLAMP1,2 UP
W65.09 BOOL  ; IND.WORK CLAMP 3 PRESS
W65.10 BOOL  ; IND.WORK CLAMP 3 UN-PRESS
W65.11 BOOL  ; IND.OIL SUPPLY
W65.12 BOOL  ; IND.JIG CHANGE OVER MIRROR
W65.13 BOOL  ; IND.JIG CHANGE OVER NORMAL
W65.14 BOOL  ; IND.N/R CHANGE OVER MIRROR
W65.15 BOOL  ; IND.N/R CHANGE OVER NORMAL
W66.00 BOOL  ; IND.WORK CLAMP CHANGE OVER MIRROR
W66.01 BOOL  ; IND.WORK CLAMP CHANGE OVER NORMAL
W66.02 BOOL  ; IND.NR START
W66.03 BOOL  ; IND.NR REV DIRECTION
W66.04 BOOL  ; IND.NR NORMAL DIRECTION
W66.05 BOOL  ; IND.NR FINISH CONF.
W67.00 BOOL  ; IND.SOL POKAYOKE PULG ASSY
W68.00 BOOL  ; IND.WPRK PUSHER DOWN
W68.01 BOOL  ; IND WORK PUSHER UP
W68.02 BOOL  ; IND MASTER CHECK ON
W68.03 BOOL  ; IND MASTER OK
W68.04 BOOL  ; IND MASTER NG
W68.05 BOOL  ; IND GD-P3S SELECTION
W68.06 BOOL  ; IND GD-P3SH SELECTION
W6.00 BOOL  ; BUZZER RESET (ALL FAULT)
W6.02 BOOL  ; BZ.RESET(PLC_BATTERY CHANGE)
W75.00 BOOL  ; AUTO CONDITION
W75.01 BOOL  ; AUTO START CONDITION
W75.02 BOOL  ; AUTO PRESET START CONDITION
W75.03 BOOL  ; AutoRunning
W75.04 BOOL  ; CYCLE_STOP
W75.05 BOOL  ; P11 AutoMotionStart
W75.06 BOOL  ; P11 AutoMotion CycleEnd
W75.07 BOOL  ; P12 AutoMotionStart
W75.08 BOOL  ; P12 AutoMotion CycleEnd
W75.09 BOOL  ; P13 AutoMotionStart
W75.10 BOOL  ; P13 AutoMotion CycleEnd
W75.11 BOOL  ; P14 AutoMotionStart
W75.12 BOOL  ; P14 AutoMotion CycleEnd
W75.13 BOOL  ; P15 AutoMotionStart
W75.14 BOOL  ; P15 AutoMotion CycleEnd
W75.15 BOOL  ; P16 AutoMotionStart
W76.00 BOOL  ; P16 AutoMotion CycleEnd
W76.01 BOOL  ; P17 AutoMotionStart
W76.02 BOOL  ; P17 AutoMotion CycleEnd
W76.03 BOOL  ; P18 AutoMotionStart
W76.04 BOOL  ; P18 AutoMotion CycleEnd
W77.00 BOOL  ; ALL NOT OPERATE
W78.04 BOOL  ; Machine Stop
W80.00 BOOL  ; AUTO START
W80.01 BOOL  ; QR-READ START OPERATION
W80.02 BOOL  ; QR-READ CONF. NORMAL
W80.03 BOOL  ; QR-READ CONF. ERROR
W80.04 BOOL  ; QR-READ FINISH
W80.05 BOOL  ; PREVIOUS M/C PROCESS SKIP CHECK
W80.06 BOOL  ; THIS M/C PROCESS COMPLETE CHECK
W80.07 BOOL  ; SKIP PROCESS DETECT
W80.08 BOOL  ; REPEAT PROCESS DETECT
W80.09 BOOL  ; CLAMP STARTING
W80.10 BOOL  ; SOL.DUMMY FRANGE CLAMP
W80.11 BOOL  ; DUMMY FRANGE CLAMP  CONF.
W80.12 BOOL  ; PLUG RELIEF NORMAL OPERATE
W80.13 BOOL  ; PLUG RELIEF MIRROR OPERATE
W80.14 BOOL  ; SOL.TIGHTENING SLIDE 2 RET.
W80.15 BOOL  ; TIGHTENING SLIDE 2 RET.CONF.
W81.00 BOOL  ; SOL.JIG CHANGE OVER MIRROR
W81.01 BOOL  ; JIG CHANGE OVER MIRROR CONF.
W81.02 BOOL  ; SOL.N/R CHANGE OVER MIRROR
W81.03 BOOL  ; N/R CHANGE OVER MIRROR CONF.
W81.04 BOOL  ; SOL.WORK CLAMP CHANGE OVER MIRROR
W81.05 BOOL  ; WORK CLAMP CHANGE OVER MIRROR CONF.
W81.06 BOOL  ; SOL.TIGHTENING SLIDE 2 RTN.
W81.07 BOOL  ; TIGHTENING SLIDE 2 RTN.CONF.
W81.08 BOOL  ; SOL.JIG CHANGE OVER NORMAL
W81.09 BOOL  ; JIG CHANGE OVER NORMAL CONF.
W81.10 BOOL  ; SOL.N/R CHANGE OVER NORMAL
W81.11 BOOL  ; N/R CHANGE OVER NORMAL CONF.
W81.12 BOOL  ; SOL.WORK CLAMP CHANGE OVER NORMAL
W81.13 BOOL  ; WORK CLAMP CHANGE OVER NORMAL CONF.
W81.14 BOOL  ; SOL.WORK CLAMP 1,2 CLAMP
W81.15 BOOL  ; WORK CLAMP 1,2 CLAMP CONF.
W82.00 BOOL  ; SOL.WORK CLAMP 3 PRESS
W82.01 BOOL  ; WORK CLAMP 3 PRESS CONF.
W82.02 BOOL  ; SOL.TIGHTENING SLIDE 1 TIGHT.
W82.03 BOOL  ; TIGHTENING SLIDE 1 TIGHT. CONF.
W82.04 BOOL  ; SOL.TIGHTENING SLIDE 2 ADV.
W82.05 BOOL  ; TIGHTENING SLIDE 2 ADV. CONF.
W82.06 BOOL  ; N/R PROCESS START
W82.07 BOOL  ; N/R PROCESS CONF.
W82.08 BOOL  ; SOL.TIGHTENING SLIDE 2 RET.
W82.09 BOOL  ; TIGHTENING SLIDE 2 RET. CONF.
W82.10 BOOL  ; SOL.TIGHTEN SLIDE 1 HOME
W82.11 BOOL  ; TIGHTEN SLIDE 1 HOME CONF.
W82.12 BOOL  ; SOL.WORK CLAMP 3 UN-PRESS
W82.13 BOOL  ; WORK CLAMP 3 UN-PRESS CONF.
W82.14 BOOL  ; ID WRITE START OPERATE
W82.15 BOOL  ; ID-WRITE CONF. NORMAL
W83.00 BOOL  ; ID-WRITE CONF. ERROR
W83.01 BOOL  ; ID-WRITE FINISH
W83.02 BOOL  ; MEMORY WRITE START OPERATE
W83.03 BOOL  ; MEMORY WRITE CONF.(FOR NEXT STEP PROGRAM)
W83.04 BOOL  ; SOL.WORK CLAMP 1,2 UN-CLAMP
W83.05 BOOL  ; WORK CLAMP 1,2 UN-CLAMP CONF.
W83.06 BOOL  ; SOL.DUMMY FRANGE UN-CLAMP
W83.07 BOOL  ; DUMMY FRANGE UN-CLAMP  CONF.
W83.08 BOOL  ; SOL.SAFETY COVER OPEN
W83.09 BOOL  ; SAFETY COVER OPEN  CONF.
W83.10 BOOL  ; ONE MC CYCLE END
W83.11 BOOL  ; ONE SHOT BEEP FOR WORK OK
W83.13 BOOL  ; MEMORY WRIT CONF.(FOR WAIT DATA)
W83.14 BOOL  ; MEMORY WRITE WAIT DATA
W83.15 BOOL  ; WAIT DATA COMPLETE
W84.00 BOOL  ; SUM CHECK NOT MATCH
W84.01 BOOL  ; PREVIOUS M/C PROCESS NG WORK
W84.02 BOOL  ; PREVIOUS M/C PROCESS UNDEFINED
W84.10 BOOL  ; PREVIOS M/C NG WORK DETECT
W84.11 BOOL  ; PREVIOS M/C UNDEFINED DETECT
W84.12 BOOL  ; P/N NOT MATCH FROM ID
W85.00 BOOL  ; 1st TORQUE CHECK -NG
W85.01 BOOL  ; 1st TORQUE CHECK OK
W85.02 BOOL  ; 1st TORQUE CHECK +NG
W85.03 BOOL  ; 1st ANGLE CHECK -NG
W85.04 BOOL  ; 1st ANGLE CHECK OK
W85.05 BOOL  ; 1st ANGLE CHECK +NG
W85.06 BOOL  ; 1st NR TIME NG(6)
W85.07 BOOL  ; 2nd TORQUE CHECK -NG
W85.08 BOOL  ; 2nd TORQUE CHECK OK
W85.09 BOOL  ; 2nd TORQUE CHECK +NG
W85.10 BOOL  ; 2nd ANGLE CHECK -NG
W85.11 BOOL  ; 2nd ANGLE CHECK OK
W85.12 BOOL  ; 2nd ANGLE CHECK +NG
W85.13 BOOL  ; IND.WORK ROTATE IN PRE-POSITION
W85.14 BOOL  ; 2nd NR TIME NG(6)
W86.00 BOOL  ; TIGHTENING RESULT RESET
W86.01 BOOL  ; WORK NG
W86.02 BOOL  ; WORK OK
W86.03 BOOL  ; NR TIME NG
W86.04 BOOL  ; FASTENING NG No.
W86.05 BOOL  ; FASTENING NG
W87.00 BOOL  ; PLUG OIL SUPPLY START MOTOR
W87.01 BOOL  ; PLUG OIL SUPPLY CONF.
W87.05 BOOL  ; CHECK PLUG MODEL CONDITION
W87.06 BOOL  ; CHECK PLUG MODEL START
W87.07 BOOL  ; PLUG MODEL GD-P3S CHECK OK
W87.08 BOOL  ; PLUG MODEL GD-P3S CHECK NG
W88.00 BOOL  ; NAGARA START
W88.01 BOOL  ; WORK PUSHER DOWN
W88.02 BOOL  ; WORK PUSHER DW CONF.
W88.03 BOOL  ; START TEST COVER
W88.04 BOOL  ; WORK PUSHER UP
W88.05 BOOL  ; WORK PUSHER UP CONF.
W88.06 BOOL  ; PUSHER UP (NG CASE)
W88.07 BOOL  ; PUSHER UP CONF. (NG CASE)
W90.00 BOOL  ; Takeout Positioning COND
W90.01 BOOL  ; Takeout MB feed  & Positioning COND
W90.02 BOOL  ; Takeout Vacum Cond
W90.03 BOOL  ; Take in VAcuum COND
W90.04 BOOL  ; Take in Vacuum & Slide COND
W90.05 BOOL  ; Take in Slide transfer Cond
W90.06 BOOL  ; Unit1CycleStartConditionAux7
W90.07 BOOL  ; Unit1CycleStartConditionAux8
W90.08 BOOL  ; Unit1CycleStartConditionAux9
W90.09 BOOL  ; P11 CycleStartCond
W90.10 BOOL  ; N/R RUNNING
W90.11 BOOL  ; START N/R CONDITION CONF.
W91.00 BOOL  ; Unit2CycleStartConditionAux1
W91.01 BOOL  ; Unit2CycleStartConditionAux2
W91.02 BOOL  ; Unit2CycleStartConditionAux3
W91.03 BOOL  ; Unit2CycleStartConditionAux4
W91.04 BOOL  ; Unit2CycleStartConditionAux5
W91.05 BOOL  ; Unit2CycleStartConditionAux6
W91.06 BOOL  ; Unit2CycleStartConditionAux7
W91.07 BOOL  ; Unit2CycleStartConditionAux8
W91.08 BOOL  ; Unit2CycleStartConditionAux9
W91.09 BOOL  ; P12 CycleStartCond
W92.00 BOOL  ; shutter 1 close condition
W92.01 BOOL  ; Unit3CycleStartConditionAux2
W92.02 BOOL  ; shutter 1 open cond
W92.03 BOOL  ; Unit3CycleStartConditionAux4
W92.04 BOOL  ; Unit3CycleStartConditionAux5
W92.05 BOOL  ; Unit3CycleStartConditionAux6
W92.06 BOOL  ; Unit3CycleStartConditionAux7
W92.07 BOOL  ; Unit3CycleStartConditionAux8
W92.08 BOOL  ; Unit3CycleStartConditionAux9
W92.09 BOOL  ; P13 CycleStartCond
W92.10 BOOL  ; 2nd ANGLE CHECK -NG STEP 2
W92.11 BOOL  ; 2nd ANGLE CHECK OK - STEP 2
W92.12 BOOL  ; 2nd ANGLE CHECK +NG STEP 2
W92.13 BOOL  ; 2nd TORQUE RATE NG - STEP 2
W92.14 BOOL  ; 2nd NR TIME NG(6) STEP 2
W92.15 BOOL  ; WORK OK JUDE STEP 2
W93.00 BOOL  ; Unit4CycleStartConditionAux1
W93.01 BOOL  ; Unit4CycleStartConditionAux2
W93.02 BOOL  ; Unit4CycleStartConditionAux3
W93.03 BOOL  ; Unit4CycleStartConditionAux4
W93.04 BOOL  ; Unit4CycleStartConditionAux5
W93.05 BOOL  ; Unit4CycleStartConditionAux6
W93.06 BOOL  ; Unit1CycleStartConditionAux7
W93.07 BOOL  ; Unit1CycleStartConditionAux8
W93.08 BOOL  ; Unit1CycleStartConditionAux9
W93.09 BOOL  ; Unit1CycleStartConditionAux10
W93.10 BOOL  ; P14 CycleStartCond
W93.15 BOOL  ; TOTAL NG STEP 2
W94.00 BOOL  ; Unit5CycleStartConditionAux1
W94.01 BOOL  ; Unit5CycleStartConditionAux2
W94.02 BOOL  ; Unit5CycleStartConditionAux3
W94.03 BOOL  ; Unit5CycleStartConditionAux4
W94.04 BOOL  ; Unit5CycleStartConditionAux5
W94.05 BOOL  ; Unit5CycleStartConditionAux6
W94.06 BOOL  ; Unit5CycleStartConditionAux7
W94.07 BOOL  ; Unit5CycleStartConditionAux8
W94.08 BOOL  ; Unit5CycleStartConditionAux9
W94.09 BOOL  ; P15 CycleStartCond
W94.10 BOOL  ; P14 CycleStartCond
W95.00 BOOL  ; Take out Raw work COND
W95.01 BOOL  ; Take In Raw Work COND
W95.02 BOOL  ; Take Out Finish Work COND
W95.03 BOOL  ; Take In Finish Work COND
W95.04 BOOL  ; Unit6CycleStartCond GP1,2 Unload FN (Discharge)
W95.05 BOOL  ; Unit6CycleStartConditionAux6
W95.06 BOOL  ; Unit6CycleStartConditionAux7
W95.07 BOOL  ; Unit6CycleStartConditionAux8
W95.08 BOOL  ; Unit6CycleStartConditionAux9
W95.09 BOOL  ; Unit6CycleStartConditionAux10
W95.10 BOOL  ; P16 Cycle StartCond
W96.00 BOOL  ; Unit7CycleStartConditionAux1
W96.01 BOOL  ; Unit7CycleStartConditionAux2
W96.02 BOOL  ; Unit7CycleStartConditionAux3
W96.03 BOOL  ; Unit7CycleStartConditionAux4
W96.04 BOOL  ; Unit7CycleStartConditionAux5
W96.05 BOOL  ; Unit7CycleStartConditionAux6
W96.06 BOOL  ; Unit7CycleStartConditionAux7
W96.07 BOOL  ; Unit7CycleStartConditionAux8
W96.08 BOOL  ; Unit7CycleStartConditionAux9
W96.09 BOOL  ; P17 CycleStartCond
W96.10 BOOL  ; P17 Cycle StartCond
W96.11 BOOL  ; HOLD DATA TORUE STEP 1
W96.15 BOOL  ; WORK OK JUDE STEP 1
W97.00 BOOL  ; Unit4CycleStartConditionAux1
W97.01 BOOL  ; Unit4CycleStartConditionAux2
W97.02 BOOL  ; Unit4CycleStartConditionAux3
W97.03 BOOL  ; Unit4CycleStartConditionAux4
W97.04 BOOL  ; Unit4CycleStartConditionAux5
W97.05 BOOL  ; Unit4CycleStartConditionAux6
W97.06 BOOL  ; Unit4CycleStartConditionAux7
W97.07 BOOL  ; Unit4CycleStartConditionAux8
W97.08 BOOL  ; Unit4CycleStartConditionAux9
W97.09 BOOL  ; Unit4CycleStartConditionAux10
W97.10 BOOL  ; P18 CycleStartCond
W98.02 BOOL  ; QR-READ CONF. NORMAL ID2
W98.03 BOOL  ; QR-READ CONF. ERROR
W98.04 BOOL  ; QR-READ FINISH ID2
W9.01 BOOL  ; COIL DESIGN. SPARE2
W9.02 BOOL  ; COIL DESIGN. SPARE3
W9.03 BOOL  ; COIL DESIGN. SPARE4
W9.04 BOOL  ; COIL DESIGN. SPARE5
W9.05 BOOL  ; COIL DESIGN. SPARE6
W9.06 BOOL  ; COIL DESIGN. SPARE7
W9.07 BOOL  ; COIL DESIGN. SPARE8
DUMMY_DOOR W100.09 BOOL  ; CR.DUMMY DOOR CONFIRM
DUMMY_DOOR_REQ W100.06 BOOL  ; PB.DUMMY DOOR OPEN REQUEST
Disch_CMD_P11 E0_0.00 BOOL
Disch_CMD_P16 E0_0.01 BOOL
Disch_compl_P11 E0_0.02 BOOL
Disch_compl_P14 E0_0.03 BOOL
Disch_compl_P15 E0_0.04 BOOL
Disch_compl_P16 E0_0.05 BOOL
Discharge_Complete E0_0.06 BOOL
Discharge_main E0_0.07 BOOL
EC1_ALARM W102.02 BOOL  ; 1EC1.ALARM
EC2_ALARM W102.05 BOOL  ; 1EC2.ALARM
EC3_ALARM W102.09 BOOL  ; 1EC3.ALARM
EC4_ALARM W102.12 BOOL  ; 1EC4.ALARM
FUSE_NORMAL W100.13 BOOL  ; CR.FUSE NORMAL CONFIRM
GB000_023 E0_46.00 BOOL  ; Trial mode
GB010_69 E0_0.08 BOOL  ; Homepos for discharge
GB011_006 E0_0.09 BOOL  ; EC1 Down allowed
GB011_007 E0_0.10 BOOL  ; SLide Request FWd
GB013_004 E0_0.11 BOOL  ; Req Slide FWD
GB014_053 E0_45.07 BOOL  ; Door 2 OPEN req
GB014_054 E0_44.14 BOOL  ; Door 2 aprrove
GB014_057 E0_44.12 BOOL  ; IND door enable req
GB014_066 E0_42.13 BOOL  ; VAcuum 1 start
GB014_069 E0_51.01 BOOL  ; oil supply
GB016_004 E0_0.12 BOOL  ; EC1 req Down
GB016_005 E0_45.10 BOOL  ; EC1 req1
GB016_006 E0_0.13 BOOL  ; Slide Forward allowed
GB016_007 E0_46.13 BOOL  ; Index table rotate allowed
GB016_008 E0_46.14 BOOL  ; EC1 down allowed
GB016_045 E0_45.11 BOOL  ; ec1 req to final caulk
GB016_068 E0_47.05 BOOL  ; Auto start trigger
GB1109 E0_0.14 BOOL  ; P11 Unit no operation
GB1199 E0_0.15 BOOL
GB1309 E0_1.00 BOOL  ; P12 unit no operation
GB1399 E0_1.01 BOOL
GB1401 E0_1.02 BOOL  ; door enable
GB1407 E0_1.03 BOOL  ; door enable
GB1409 E0_1.04 BOOL  ; P13 no operation
GB1599 E0_1.05 BOOL
GB1709 E0_1.06 BOOL  ; P14 no operation
GB1799 E0_1.08 BOOL
GB1909 E0_1.09 BOOL  ; P15 No operation
GB1999 E0_1.10 BOOL
GB2109 E0_1.11 BOOL  ; P16 no operation
GB2199 E0_1.12 BOOL
GB2309 E0_1.13 BOOL  ; P17 No operation
GB2399 E0_1.14 BOOL
GB2401 E0_1.15 BOOL
GB2403 E0_2.00 BOOL  ; 1EC3 MIDWARD START
GB24031 E0_2.01 BOOL  ; LB24031
GB2405 E0_2.02 BOOL
GB2407 E0_2.03 BOOL
GB2409 E0_2.04 BOOL
GB2411 E0_2.05 BOOL
GB2414 E0_2.06 BOOL
GB2416 E0_2.07 BOOL  ; 1EC3 MIDWARD MID START
GB24161 E0_2.08 BOOL  ; $?St$Bk?_#[3001] / 1EC3 BACKWARD START / 1EC3 BACKWARD START$?St$Bk?_#[3001]
GB2418 E0_2.09 BOOL
GB2420 E0_2.10 BOOL
GB2422 E0_2.11 BOOL
GB2425 E0_2.12 BOOL
GB2427 E0_2.13 BOOL  ; 1EC3 FORWARD START
GB2429 E0_2.14 BOOL
GB2431 E0_2.15 BOOL
GB2433 E0_3.00 BOOL
GB2435 E0_3.01 BOOL
GB2437 E0_3.02 BOOL  ; 1EC3 BACKWARD START
GB2440 E0_3.03 BOOL
GB2442 E0_3.04 BOOL  ; 1EC3 FORWARD START
GB2444 E0_3.05 BOOL
GB2446 E0_3.06 BOOL
GB2448 E0_3.07 BOOL
GB2450 E0_3.08 BOOL  ; 1EC3 BACKWARD START
GB2599 E0_3.09 BOOL
GB7509 E0_43.13 BOOL  ; P13_1 AutoMotionStart
GB7510 E0_43.15 BOOL  ; P13a cycle END
GSB000 W0.00 BOOL  ; FOR EQUIPMENT DESIGN_ORDINARY TIMES ON
GSB001 W0.01 BOOL  ; FOR EQUIPMENT DESIGN_ORDINARY TIMES OFF
GSB002 W0.02 BOOL  ; FOR EQUIPMENT DESIGN_1EC3 MID ELIMINED MODIF BY MCH
GSB003 W0.03 BOOL  ; FOR EQUIPMENT DESIGN_ORDINARY TIMES OFF_2
GSB004 W0.04 BOOL  ; FOR EQUIPMENT DESIGN_ORDINARY TIMES OFF_3
GSB005 W0.05 BOOL  ; FOR EQUIPMENT DESIGN_ORDINARY TIMES OFF_4
GSB006 W0.06 BOOL  ; FOR EQUIPMENT DESIGN_ORDINARY TIMES OFF_5
GSB007 W0.07 BOOL  ; FOR EQUIPMENT DESIGN_ORDINARY TIMES OFF_6
GSB008 W0.08 BOOL  ; FOR EQUIPMENT DESIGN_ORDINARY TIMES OFF_7
GT367 T3032 TIMER  ; trigger cover open
LB450 E0_1.07 BOOL  ; IND 1 cycle
LS_3301_00 W150.00 BOOL  ; SHUTTER 1 UP CONFIRM
LS_3301_01 W150.01 BOOL  ; AS.SHUTTER 1 DOOR DOWN CONFIRM
LS_3301_02 W150.02 BOOL  ; AS.SHUTTER 2  UP CONFIRM
LS_3301_03 W150.03 BOOL  ; SHUTTER 2 DOWN CONFIRM
LS_3301_04 W150.04 BOOL  ; AS.GRIPPER UNIT DOWN CONFIRM
LS_3301_05 W150.05 BOOL  ; AS.GRIPPER UNIT UP CONFIRM
LS_3301_06 W150.06 BOOL  ; AS.GRIPPER 1 DIAPH CHUCK. CONFIRM
LS_3301_07 W150.07 BOOL  ; AS.GRIPPER 1 DIAPH UNCHUCK. CONFIRM
LS_3301_08 W150.08 BOOL  ; AS.GRIPPER 2 DIAPH CHUCK. CONFIRM
LS_3301_09 W150.09 BOOL  ; AS.GRIPPER 2 DIAPH UNCHUCK. CONFIRM
LS_3301_10 W150.10 BOOL  ; AS.GRIPPER 3 DIAPH CHUCK. CONFIRM
LS_3301_11 W150.11 BOOL  ; AS.GRIPPER 3 DIAPH UNCHUCK. CONFIRM
LS_3301_12 W150.12 BOOL  ; AS.FLIP DIAPH 180. CONFIRM
LS_3301_13 W150.13 BOOL  ; AS.FLIP DIAPH 0. CONFIRM
LS_3301_15_START W150.15 BOOL  ; AUTO START(NAGARA)
LS_3302_00 W151.00 BOOL  ; AS.GIPPER TRANSFER 1 UNIT CHUCK CONFIRM
LS_3302_01 W151.01 BOOL  ; AS.GIPPER TRANSFER 1 UNIT  UNCHUCK CONFIRM
LS_3302_02 W151.02 BOOL  ; AS.GIPPER TRANSFER 2 UNIT CHUCK CONFIRM
LS_3302_03 W151.03 BOOL  ; AS.GIPPER TRANSFER 2 UNIT  UNCHUCK CONFIRM
LS_3302_04 W151.04 BOOL  ; AS.GIPPER TRANSFER UNIT 1 UNIT ADV. CONFIRM
LS_3302_05 W151.05 BOOL  ; AS.GIPPER TRANSFER UNIT 1 UNIT RET. CONFIRM
LS_3302_06 W151.06 BOOL  ; AS.GIPPER TRANSFER UNIT 2 UNIT ADV. CONFIRM
LS_3302_07 W151.07 BOOL  ; AS.GIPPER TRANSFER UNIT 2 UNIT RET. CONFIRM
LS_3303_00 W152.00 BOOL  ; AS.M&B LOAD IN DOWN.CONFIRM
LS_3303_01 W152.01 BOOL  ; AS.M&B LOAD IN UP.CONFIRM
LS_3303_02 W152.02 BOOL  ; AS.M&B LOAD OUT DOWN.CONFIRM
LS_3303_03 W152.03 BOOL  ; AS.M&B LOAD OUT UP.CONFIRM
LS_3303_04 W152.04 BOOL  ; AS.M&B LOAD OUT UNIT DOWN.CONFIRM
LS_3303_05 W152.05 BOOL  ; AS.M&B LOAD OUT UNIT UP.CONFIRM
LS_3303_06 W152.06 BOOL  ; AS.M&B LOAD UNIT SLIDE ADV.CONFIRM
LS_3303_07 W152.07 BOOL  ; AS.M&B LOAD UNIT SLIDE RET.CONFIRM
LS_3303_08 W152.08 BOOL  ; AS.PIN POSIRIONNING UP CONFIRM
LS_3303_09 W152.09 BOOL  ; AS.PIN POSIRIONNING DOWN CONFIRM
LS_3303_10 W152.10 BOOL  ; AS.TRANSFER SLIDE UNIT ADV. CONFIRM
LS_3303_11 W152.11 BOOL  ; AS.TRANSFER SLIDE UNIT RET. CONFIRM
LS_3303_14 E0_46.11 BOOL  ; AS LOAD BWD
LS_3303_15 E0_47.11 BOOL  ; LS LOAD IN FWD
LS_3304_00 W153.00 BOOL  ; AS.WORK FINISH TRAY DOWN CONFIRM
LS_3304_01 W153.01 BOOL  ; AS.WORK FINISH TRAY UP CONFIRM
LS_3304_02 W153.02 BOOL  ; AS.OK PUSH UP. CONFIRM
LS_3304_03 W153.03 BOOL  ; AS.OK PUSH DOWN. CONFIRM
LS_3304_04 W153.04 BOOL  ; AS.NG PULL DOWN. CONFIRM
LS_3304_05 W153.05 BOOL  ; AS.NG PUSH UP. CONFIRM
LS_EC1_BACKWARD W102.01 BOOL  ; 1EC1.BACKWARD COMPLETE
LS_EC1_FORWARD W102.00 BOOL  ; 1EC1.FORWARD COMPLETE
LS_EC2_BACKWARD W102.04 BOOL  ; 1EC2.BACKWARD COMPLETE
LS_EC2_FORWARD W102.03 BOOL  ; 1EC2.FORWARD COMPLETE
LS_EC3_BACKWARD W102.07 BOOL  ; 1EC3.BACKWARD COMPLETE
LS_EC3_FORWARD W102.06 BOOL  ; 1EC3.FORWARD COMPLETE
LS_EC4_BACKWARD W102.11 BOOL  ; 1EC4.BACKWARD COMPLETE
LS_EC4_FORWARD W102.10 BOOL  ; 1EC4.FORWARD COMPLETE
MOTOR_ALARM W150.14 BOOL  ; 1MTD1.ALARM
MSTR_RDY W100.12 BOOL  ; CR.MASTER ON CONFIRM
PB_AUTORUN W100.04 BOOL  ; PB.AUTO RUN
PB_CYCLE_STOP W100.05 BOOL  ; PB.CYCLE STOP
PB_EMG_NOT W100.00 BOOL  ; PB.EMERGENCY STOP NOT OPERATE
PB_MASTER_ON W100.03 BOOL  ; PB.MASTER ON
PH_3302_08_OFF W154.08 BOOL  ; PH. DUMMY FEED IN CONFIRM off
PH_3302_08_OFFF W156.07 BOOL  ; PH. MB FEED IN CONFIRM off
PH_3302_08_ON W151.08 BOOL  ; PH. DUMMY FEED IN CONFIRM on
